# B&R Automation Studio project Parker_BMM_ST_V5_3147_V12 (part 32)

#### ClampR.ax
```
InitParameter (Version=5.06.1, NcSwId=ACP10)
  ACP10AXIS_typ:
    dig_in:
      level:
        reference = ncACTIV_HI
        pos_hw_end = ncACTIV_HI
        neg_hw_end = ncACTIV_HI
        trigger1 = ncACTIV_HI
        trigger2 = ncACTIV_HI + ncQUICKSTOP
    encoder_if:
      parameter:
        count_dir = ncSTANDARD
        scaling:
          load:
            units = 7087
            rev_motor = 5
    limit:
      parameter:
        v_pos = 70870.0  // Speed in positive direction    5600rpm 120000   4000rpm 85600
        v_neg = 70870.0
        a1_pos = 472400.0
        a2_pos = 472400.0
        a1_neg = 472400.0
        a2_neg = 472400.0
        t_jolt = 0.1
        t_in_pos = 0.0
        pos_sw_end = 8388607
        neg_sw_end = -8388608
        ds_warning = 354.0
        ds_stop = 708.0
        a_stop = 1.0E+30
        dv_stop = 0.0
        dv_stop_mode = ncOFF
    controller:
      mode = ncPOSITION
      position:
        kv = 66.0
        tn = 0.0
        t_predict = 0.0004
        t_total = 0.0004
        p_max = 1.0E+30
        i_max = 0.0
      speed:
        kv = 6.4
        tn = 0.1  // Integral action time 0.1
        t_filter = 0.0048  // Filter time constant 0.0048
        isq_filter1:
          type = ncOFF
          a0 = 0.0
          a1 = 0.0
          b0 = 0.0
          b1 = 0.0
          b2 = 0.0
          c0_par_id = 0
          c1_par_id = 0
        isq_filter2:
          type = ncOFF
          a0 = 0.0
          a1 = 0.0
          b0 = 0.0
          b1 = 0.0
          b2 = 0.0
          c0_par_id = 0
          c1_par_id = 0
        isq_filter3:
          type = ncOFF
          a0 = 0.0
          a1 = 0.0
          b0 = 0.0
          b1 = 0.0
          b2 = 0.0
          c0_par_id = 0
          c1_par_id = 0
      uf:
        type = ncLINEAR
        auto_config = ncMOTOR_PAR
        u0 = 0.0
        un = 0.0
        fn = 50.0
        k_f_slip = 0.0
      ff:
        mode = ncSTANDARD
        torque_load = 0.0
        torque_pos = 0.0
        torque_neg = 0.0
        kv_torque = 0.0
        inertia = 0.0
        t_filter_a = 0.0
      fb:
        mode = ncSTANDARD
        speed_mix_ratio = 0.0
        speed_kv = 2.0
      model:
        mass1:
          inertia = 0
          viscous_friction = 0
        mass2:
          inertia = 0
          viscous_friction = 0
          stiffness = 0
          damping = 0
    move:
      stop:
        parameter[0]:
          decel_ramp = ncA_LIMIT
          controller = ncON
        parameter[1]:
          decel_ramp = ncA_LIMIT
          controller = ncON
        parameter[2]:
          decel_ramp = ncA_LIMIT
          controller = ncON
        parameter[3]:
          decel_ramp = ncA_LIMIT
          controller = ncON
        quickstop:
          decel_ramp = ncA_LIMIT
          t_jolt = 0
        drive_error:
          decel_ramp = ncA_LIMIT
      homing:
        parameter:
          s = 0
          v_switch = 5000.0
          v_trigger = 500.0
          a = 50000.0
          mode = ncDIRECT
          edge_sw = ncPOSITIVE
          start_dir = ncPOSITIVE
          trigg_dir = ncPOSITIVE
          ref_pulse = ncOFF
          fix_dir = ncOFF
          tr_s_block = 0.0
          torque_lim = 0.0
          ds_block = 0.0
          ds_stop = 0.0
      basis:
        parameter:
          v_pos = 500.0
          v_neg = 500.0
          a1_pos = 5000.0
          a2_pos = 5000.0
          a1_neg = 5000.0
          a2_neg = 5000.0
    message:
      text:
        parameter:
          format = ncBREAK
          columns = 80
          data_modul = acp10etxen
```

### Data object Logical/Motion/init/ClampL (Ax)

#### ClampL.ax
```
InitParameter (Version=5.06.1, NcSwId=ACP10)
  ACP10AXIS_typ:
    dig_in:
      level:
        reference = ncACTIV_HI
        pos_hw_end = ncACTIV_HI
        neg_hw_end = ncACTIV_HI
        trigger1 = ncACTIV_HI
        trigger2 = ncACTIV_HI + ncQUICKSTOP
    encoder_if:
      parameter:
        count_dir = ncSTANDARD
        scaling:
          load:
            units = 1495
            rev_motor = 1
    limit:
      parameter:
        v_pos = 74750.0  // Speed in positive direction    5600rpm 120000   4000rpm 85600
        v_neg = 74750.0
        a1_pos = 747500.0
        a2_pos = 747500.0
        a1_neg = 747500.0
        a2_neg = 747500.0
        t_jolt = 0.1
        t_in_pos = 0.0
        pos_sw_end = 8388607
        neg_sw_end = -8388608
        ds_warning = 325.0
        ds_stop = 750.0
        a_stop = 1.0E+30
        dv_stop = 0.0
        dv_stop_mode = ncOFF
    controller:
      mode = ncPOSITION
      position:
        kv = 210.0
        tn = 0.0
        t_predict = 0.0004
        t_total = 0.0004
        p_max = 1.0E+30
        i_max = 0.0
      speed:
        kv = 15.0
        tn = 0.1  // Integral action time 0.1
        t_filter = 0.0048  // Filter time constant 0.0048
        isq_filter1:
          type = ncOFF
          a0 = 0.0
          a1 = 0.0
          b0 = 0.0
          b1 = 0.0
          b2 = 0.0
          c0_par_id = 0
          c1_par_id = 0
        isq_filter2:
          type = ncOFF
          a0 = 0.0
          a1 = 0.0
          b0 = 0.0
          b1 = 0.0
          b2 = 0.0
          c0_par_id = 0
          c1_par_id = 0
        isq_filter3:
          type = ncOFF
          a0 = 0.0
          a1 = 0.0
          b0 = 0.0
          b1 = 0.0
          b2 = 0.0
          c0_par_id = 0
          c1_par_id = 0
      uf:
        type = ncLINEAR
        auto_config = ncMOTOR_PAR
        u0 = 0.0
        un = 0.0
        fn = 50.0
        k_f_slip = 0.0
      ff:
        mode = ncSTANDARD
        torque_load = 0.0
        torque_pos = 0.0
        torque_neg = 0.0
        kv_torque = 0.0
        inertia = 0.0
        t_filter_a = 0.0
      fb:
        mode = ncSTANDARD
        speed_mix_ratio = 0.0
        speed_kv = 2.0
      model:
        mass1:
          inertia = 0
          viscous_friction = 0
        mass2:
          inertia = 0
          viscous_friction = 0
          stiffness = 0
          damping = 0
    move:
      stop:
        parameter[0]:
          decel_ramp = ncA_LIMIT
          controller = ncON
        parameter[1]:
          decel_ramp = ncA_LIMIT
          controller = ncON
        parameter[2]:
          decel_ramp = ncA_LIMIT
          controller = ncON
        parameter[3]:
          decel_ramp = ncA_LIMIT
          controller = ncON
        quickstop:
          decel_ramp = ncA_LIMIT
          t_jolt = 0
        drive_error:
          decel_ramp = ncA_LIMIT
      homing:
        parameter:
          s = 0
          v_switch = 5000.0
          v_trigger = 500.0
          a = 50000.0
          mode = ncDIRECT
          edge_sw = ncPOSITIVE
          start_dir = ncPOSITIVE
          trigg_dir = ncPOSITIVE
          ref_pulse = ncOFF
          fix_dir = ncOFF
          tr_s_block = 0.0
          torque_lim = 0.0
          ds_block = 0.0
          ds_stop = 0.0
      basis:
        parameter:
          v_pos = 500.0
          v_neg = 500.0
          a1_pos = 5000.0
          a2_pos = 5000.0
          a1_neg = 5000.0
          a2_neg = 5000.0
    message:
      text:
        parameter:
          format = ncBREAK
          columns = 80
          data_modul = acp10etxen
```

### Data object Logical/Motion/init/CarriageR (Ax)

#### CarriageR.ax
```
InitParameter (Version=5.06.1, NcSwId=ACP10)
  ACP10AXIS_typ:
    dig_in:
      level:
        reference = ncACTIV_HI
        pos_hw_end = ncACTIV_HI
        neg_hw_end = ncACTIV_HI
        trigger1 = ncACTIV_HI
        trigger2 = ncACTIV_HI + ncQUICKSTOP
    encoder_if:
      parameter:
        count_dir = ncSTANDARD
        scaling:
          load:
            units = 2571
            rev_motor = 2
    limit:
      parameter:
        v_pos = 96410.0
        v_neg = 96410.0
        a1_pos = 964100.0
        a2_pos = 964100.0
        a1_neg = 964100.0
        a2_neg = 964100.0
        t_jolt = 0.1
        t_in_pos = 0.0
        pos_sw_end = 8388607
        neg_sw_end = -8388608
        ds_warning = 320.0
        ds_stop = 640.0
        a_stop = 1.0E+30
        dv_stop = 0.0
        dv_stop_mode = ncOFF
    controller:
      mode = ncPOSITION
      position:
        kv = 190.0
        tn = 0.0
        t_predict = 0.0004
        t_total = 0.0004
        p_max = 1.0E+30
        i_max = 0.0
      speed:
        kv = 7.8
        tn = 0.0
        t_filter = 0.0
        isq_filter1:
          type = ncOFF
          a0 = 0.0
          a1 = 0.0
          b0 = 0.0
          b1 = 0.0
          b2 = 0.0
          c0_par_id = 0
          c1_par_id = 0
        isq_filter2:
          type = ncOFF
          a0 = 0.0
          a1 = 0.0
          b0 = 0.0
          b1 = 0.0
          b2 = 0.0
          c0_par_id = 0
          c1_par_id = 0
        isq_filter3:
          type = ncOFF
          a0 = 0.0
          a1 = 0.0
          b0 = 0.0
          b1 = 0.0
          b2 = 0.0
          c0_par_id = 0
          c1_par_id = 0
      uf:
        type = ncLINEAR
        auto_config = ncMOTOR_PAR
        u0 = 0.0
        un = 0.0
        fn = 50.0
        k_f_slip = 0.0
      ff:
        mode = ncSTANDARD
        torque_load = 0.0
        torque_pos = 0.0
        torque_neg = 0.0
        kv_torque = 0.0
        inertia = 0.0
        t_filter_a = 0.0
      fb:
        mode = ncSTANDARD
        speed_mix_ratio = 0.0
        speed_kv = 2.0
      model:
        mass1:
          inertia = 0
          viscous_friction = 0
        mass2:
          inertia = 0
          viscous_friction = 0
          stiffness = 0
          damping = 0
    move:
      stop:
        parameter[0]:
          decel_ramp = ncA_LIMIT
          controller = ncON
        parameter[1]:
          decel_ramp = ncA_LIMIT
          controller = ncON
        parameter[2]:
          decel_ramp = ncA_LIMIT
          controller = ncON
        parameter[3]:
          decel_ramp = ncA_LIMIT
          controller = ncON
        quickstop:
          decel_ramp = ncA_LIMIT
          t_jolt = 0
        drive_error:
          decel_ramp = ncA_LIMIT
      homing:
        parameter:
          s = 0
          v_switch = 5000.0
          v_trigger = 500.0
          a = 50000.0
          mode = ncDIRECT
          edge_sw = ncPOSITIVE
          start_dir = ncPOSITIVE
          trigg_dir = ncPOSITIVE
          ref_pulse = ncOFF
          fix_dir = ncOFF
          tr_s_block = 0.0
          torque_lim = 0.0
          ds_block = 0.0
          ds_stop = 0.0
      basis:
        parameter:
          v_pos = 5000.0
          v_neg = 5000.0
          a1_pos = 50000.0
          a2_pos = 50000.0
          a1_neg = 50000.0
          a2_neg = 50000.0
    message:
      text:
        parameter:
          format = ncBREAK
          columns = 80
          data_modul = acp10etxen
```

### Data object Logical/Motion/init/CarriageL (Ax)

#### CarriageL.ax
```
InitParameter (Version=5.06.1, NcSwId=ACP10)
  ACP10AXIS_typ:
    dig_in:
      level:
        reference = ncACTIV_HI
        pos_hw_end = ncACTIV_HI
        neg_hw_end = ncACTIV_HI
        trigger1 = ncACTIV_HI
        trigger2 = ncACTIV_HI + ncQUICKSTOP
    encoder_if:
      parameter:
        count_dir = ncSTANDARD
        scaling:
          load:
            units = 1433
            rev_motor = 1
    limit:
      parameter:
        v_pos = 107475.0
        v_neg = 107475.0
        a1_pos = 1074750.0
        a2_pos = 1074750.0
        a1_neg = 1074750.0
        a2_neg = 1074750.0
        t_jolt = 0.1
        t_in_pos = 0.0
        pos_sw_end = 8388607
        neg_sw_end = -8388608
        ds_warning = 716.0
        ds_stop = 360.0
        a_stop = 1.0E+30
        dv_stop = 0.0
        dv_stop_mode = ncOFF
    controller:
      mode = ncPOSITION
      position:
        kv = 50.0
        tn = 0.0
        t_predict = 0.0004
        t_total = 0.0004
        p_max = 1.0E+30
        i_max = 0.0
      speed:
        kv = 2.0
        tn = 0.0
        t_filter = 0.0
        isq_filter1:
          type = ncOFF
          a0 = 0.0
          a1 = 0.0
          b0 = 0.0
          b1 = 0.0
          b2 = 0.0
          c0_par_id = 0
          c1_par_id = 0
        isq_filter2:
          type = ncOFF
          a0 = 0.0
          a1 = 0.0
          b0 = 0.0
          b1 = 0.0
          b2 = 0.0
          c0_par_id = 0
          c1_par_id = 0
        isq_filter3:
          type = ncOFF
          a0 = 0.0
          a1 = 0.0
          b0 = 0.0
          b1 = 0.0
          b2 = 0.0
          c0_par_id = 0
          c1_par_id = 0
      uf:
        type = ncLINEAR
        auto_config = ncMOTOR_PAR
        u0 = 0.0
        un = 0.0
        fn = 50.0
        k_f_slip = 0.0
      ff:
        mode = ncSTANDARD
        torque_load = 0.0
        torque_pos = 0.0
        torque_neg = 0.0
        kv_torque = 0.0
        inertia = 0.0
        t_filter_a = 0.0
      fb:
        mode = ncSTANDARD
        speed_mix_ratio = 0.0
        speed_kv = 2.0
      model:
        mass1:
          inertia = 0
          viscous_friction = 0
        mass2:
          inertia = 0
          viscous_friction = 0
          stiffness = 0
          damping = 0
    move:
      stop:
        parameter[0]:
          decel_ramp = ncA_LIMIT
          controller = ncON
        parameter[1]:
          decel_ramp = ncA_LIMIT
          controller = ncON
        parameter[2]:
          decel_ramp = ncA_LIMIT
          controller = ncON
        parameter[3]:
          decel_ramp = ncA_LIMIT
          controller = ncON
        quickstop:
          decel_ramp = ncA_LIMIT
          t_jolt = 0
        drive_error:
          decel_ramp = ncA_LIMIT
      homing:
        parameter:
          s = 0
          v_switch = 5000.0
          v_trigger = 500.0
          a = 50000.0
          mode = ncDIRECT
          edge_sw = ncPOSITIVE
          start_dir = ncPOSITIVE
          trigg_dir = ncPOSITIVE
          ref_pulse = ncOFF
          fix_dir = ncOFF
          tr_s_block = 0.0
          torque_lim = 0.0
          ds_block = 0.0
          ds_stop = 0.0
      basis:
        parameter:
          v_pos = 1000.0
          v_neg = 1000.0
          a1_pos = 50000.0
          a2_pos = 50000.0
          a1_neg = 50000.0
          a2_neg = 50000.0
    message:
      text:
        parameter:
          format = ncBREAK
          columns = 80
          data_modul = acp10etxen
```

### Data object Logical/Motion/init/BlowPinR (Ax)

#### BlowPinR.ax
```
InitParameter (Version=5.06.1, NcSwId=ACP10)
  ACP10AXIS_typ:
    dig_in:
      level:
        reference = ncACTIV_HI
        pos_hw_end = ncACTIV_HI
        neg_hw_end = ncACTIV_HI
        trigger1 = ncACTIV_HI
        trigger2 = ncACTIV_HI + ncQUICKSTOP
    encoder_if:
      parameter:
        count_dir = ncSTANDARD
        scaling:
          load:
            units = 2000
            rev_motor = 1
    limit:
      parameter:
        v_pos = 65000.0
        v_neg = 65000.0
        a1_pos = 1500000.0
        a2_pos = 1500000.0
        a1_neg = 1500000.0
        a2_neg = 1500000.0
        t_jolt = 0.1
        t_in_pos = 0.0
        pos_sw_end = 8388607
        neg_sw_end = -8388608
        ds_warning = 500.0
        ds_stop = 1000.0
        a_stop = 1.0E+30
        dv_stop = 0.0
        dv_stop_mode = ncOFF
    controller:
      mode = ncPOSITION
      position:
        kv = 135.0
        tn = 0.0
        t_predict = 0.0004
        t_total = 0.0004
        p_max = 1.0E+30
        i_max = 0.0
      speed:
        kv = 1.0
        tn = 0.0
        t_filter = 0.0
        isq_filter1:
          type = ncOFF
          a0 = 0.0
          a1 = 0.0
          b0 = 0.0
          b1 = 0.0
          b2 = 0.0
          c0_par_id = 0
          c1_par_id = 0
        isq_filter2:
          type = ncOFF
          a0 = 0.0
          a1 = 0.0
          b0 = 0.0
          b1 = 0.0
          b2 = 0.0
          c0_par_id = 0
          c1_par_id = 0
        isq_filter3:
          type = ncOFF
          a0 = 0.0
          a1 = 0.0
          b0 = 0.0
          b1 = 0.0
          b2 = 0.0
          c0_par_id = 0
          c1_par_id = 0
      uf:
        type = ncLINEAR
        auto_config = ncMOTOR_PAR
        u0 = 0.0
        un = 0.0
        fn = 50.0
        k_f_slip = 0.0
      ff:
        mode = ncSTANDARD
        torque_load = 0.0
        torque_pos = 0.0
        torque_neg = 0.0
        kv_torque = 0.0
        inertia = 0.0
        t_filter_a = 0.0
      fb:
        mode = ncSTANDARD
        speed_mix_ratio = 0.0
        speed_kv = 0.0
      model:
        mass1:
          inertia = 0.0
          viscous_friction = 0.0
        mass2:
          inertia = 0.0
          viscous_friction = 0.0
          stiffness = 0.0
          damping = 0.0
    move:
      stop:
        parameter[0]:
          decel_ramp = ncA_LIMIT
          controller = ncON
        parameter[1]:
          decel_ramp = ncA_LIMIT
          controller = ncON
        parameter[2]:
          decel_ramp = ncA_LIMIT
          controller = ncON
        parameter[3]:
          decel_ramp = ncA_LIMIT
          controller = ncON
        quickstop:
          decel_ramp = ncA_LIMIT
          t_jolt = 0.0
        drive_error:
          decel_ramp = ncA_LIMIT
      homing:
        parameter:
          s = 0
          v_switch = 5000.0
          v_trigger = 500.0
          a = 50000.0
          mode = ncDIRECT
          edge_sw = ncPOSITIVE
          start_dir = ncPOSITIVE
          trigg_dir = ncPOSITIVE
          ref_pulse = ncOFF
          fix_dir = ncOFF
          tr_s_block = 0.0
          torque_lim = 0.0
          ds_block = 0.0
          ds_stop = 0.0
      basis:
        parameter:
          v_pos = 5000.0
          v_neg = 5000.0
          a1_pos = 50000.0
          a2_pos = 50000.0
          a1_neg = 50000.0
          a2_neg = 50000.0
    message:
      text:
        parameter:
          format = ncBREAK
          columns = 80
          data_modul = acp10etxen
```

### Data object Logical/Motion/init/BlowPinL (Ax)

#### BlowPinL.ax
```
InitParameter (Version=5.06.1, NcSwId=ACP10)
  ACP10AXIS_typ:
    dig_in:
      level:
        reference = ncACTIV_HI
        pos_hw_end = ncACTIV_HI
        neg_hw_end = ncACTIV_HI
        trigger1 = ncACTIV_HI
        trigger2 = ncACTIV_HI + ncQUICKSTOP
    encoder_if:
      parameter:
        count_dir = ncSTANDARD
        scaling:
          load:
            units = 2000
            rev_motor = 1
    limit:
      parameter:
        v_pos = 65000.0
        v_neg = 65000.0
        a1_pos = 1500000.0
        a2_pos = 1500000.0
        a1_neg = 1500000.0
        a2_neg = 1500000.0
        t_jolt = 0.1
        t_in_pos = 0.0
        pos_sw_end = 8388607
        neg_sw_end = -8388608
        ds_warning = 500.0
        ds_stop = 1000.0
        a_stop = 1.0E+30
        dv_stop = 0.0
        dv_stop_mode = ncOFF
    controller:
      mode = ncPOSITION
      position:
        kv = 170.0
        tn = 0.0
        t_predict = 0.0004
        t_total = 0.0004
        p_max = 1.0E+30
        i_max = 0.0
      speed:
        kv = 3.25
        tn = 0.0
        t_filter = 0.0
        isq_filter1:
          type = ncOFF
          a0 = 0.0
          a1 = 0.0
          b0 = 0.0
          b1 = 0.0
          b2 = 0.0
          c0_par_id = 0
          c1_par_id = 0
        isq_filter2:
          type = ncOFF
          a0 = 0.0
          a1 = 0.0
          b0 = 0.0
          b1 = 0.0
          b2 = 0.0
          c0_par_id = 0
          c1_par_id = 0
        isq_filter3:
          type = ncOFF
          a0 = 0.0
          a1 = 0.0
          b0 = 0.0
          b1 = 0.0
          b2 = 0.0
          c0_par_id = 0
          c1_par_id = 0
      uf:
        type = ncLINEAR
        auto_config = ncMOTOR_PAR
        u0 = 0.0
        un = 0.0
        fn = 50.0
        k_f_slip = 0.0
      ff:
        mode = ncSTANDARD
        torque_load = 0.0
        torque_pos = 0.0
        torque_neg = 0.0
        kv_torque = 0.0
        inertia = 0.0
        t_filter_a = 0.0
      fb:
        mode = ncSTANDARD
        speed_mix_ratio = 0.0
        speed_kv = 2.0
      model:
        mass1:
          inertia = 0
          viscous_friction = 0
        mass2:
          inertia = 0
          viscous_friction = 0
          stiffness = 0
          damping = 0
    move:
      stop:
        parameter[0]:
          decel_ramp = ncA_LIMIT
          controller = ncON
        parameter[1]:
          decel_ramp = ncA_LIMIT
          controller = ncON
        parameter[2]:
          decel_ramp = ncA_LIMIT
          controller = ncON
        parameter[3]:
          decel_ramp = ncA_LIMIT
          controller = ncON
        quickstop:
          decel_ramp = ncA_LIMIT
          t_jolt = 0
        drive_error:
          decel_ramp = ncA_LIMIT
      homing:
        parameter:
          s = 0
          v_switch = 5000.0
          v_trigger = 500.0
          a = 50000.0
          mode = ncDIRECT
          edge_sw = ncPOSITIVE
          start_dir = ncPOSITIVE
          trigg_dir = ncPOSITIVE
          ref_pulse = ncOFF
          fix_dir = ncOFF
          tr_s_block = 0.0
          torque_lim = 0.0
          ds_block = 0.0
          ds_stop = 0.0
      basis:
        parameter:
          v_pos = 500.0
          v_neg = 500.0
          a1_pos = 50000.0
          a2_pos = 50000.0
          a1_neg = 50000.0
          a2_neg = 50000.0
    message:
      text:
        parameter:
          format = ncBREAK
          columns = 80
          data_modul = acp10etxen
```

### Data object Logical/Motion/init/BlowPin2R (Ax)

#### BlowPinR.ax
```
InitParameter (Version=5.06.1, NcSwId=ACP10)
  ACP10AXIS_typ:
    dig_in:
      level:
        reference = ncACTIV_HI
        pos_hw_end = ncACTIV_HI
        neg_hw_end = ncACTIV_HI
        trigger1 = ncACTIV_HI
        trigger2 = ncACTIV_HI + ncQUICKSTOP
    encoder_if:
      parameter:
        count_dir = ncSTANDARD
        scaling:
          load:
            units = 2000
            rev_motor = 1
    limit:
      parameter:
        v_pos = 65000.0
        v_neg = 65000.0
        a1_pos = 1500000.0
        a2_pos = 1500000.0
        a1_neg = 1500000.0
        a2_neg = 1500000.0
        t_jolt = 0.1
        t_in_pos = 0.0
        pos_sw_end = 8388607
        neg_sw_end = -8388608
        ds_warning = 500.0
        ds_stop = 1000.0
        a_stop = 1.0E+30
        dv_stop = 0.0
        dv_stop_mode = ncOFF
    controller:
      mode = ncPOSITION
      position:
        kv = 213.0
        tn = 0.0
        t_predict = 0.0004
        t_total = 0.0004
        p_max = 1.0E+30
        i_max = 0.0
      speed:
        kv = 2.7
        tn = 0.0
        t_filter = 0.0
        isq_filter1:
          type = ncOFF
          a0 = 0.0
          a1 = 0.0
          b0 = 0.0
          b1 = 0.0
          b2 = 0.0
          c0_par_id = 0
          c1_par_id = 0
        isq_filter2:
          type = ncOFF
          a0 = 0.0
          a1 = 0.0
          b0 = 0.0
          b1 = 0.0
          b2 = 0.0
          c0_par_id = 0
          c1_par_id = 0
        isq_filter3:
          type = ncOFF
          a0 = 0.0
          a1 = 0.0
          b0 = 0.0
          b1 = 0.0
          b2 = 0.0
          c0_par_id = 0
          c1_par_id = 0
      uf:
        type = ncLINEAR
        auto_config = ncMOTOR_PAR
        u0 = 0.0
        un = 0.0
        fn = 50.0
        k_f_slip = 0.0
      ff:
        mode = ncSTANDARD
        torque_load = 0.0
        torque_pos = 0.0
        torque_neg = 0.0
        kv_torque = 0.0
        inertia = 0.0
        t_filter_a = 0.0
      fb:
        mode = ncSTANDARD
        speed_mix_ratio = 0.0
        speed_kv = 0.0
      model:
        mass1:
          inertia = 0.0
          viscous_friction = 0.0
        mass2:
          inertia = 0.0
          viscous_friction = 0.0
          stiffness = 0.0
          damping = 0.0
    move:
      stop:
        parameter[0]:
          decel_ramp = ncA_LIMIT
          controller = ncON
        parameter[1]:
          decel_ramp = ncA_LIMIT
          controller = ncON
        parameter[2]:
          decel_ramp = ncA_LIMIT
          controller = ncON
        parameter[3]:
          decel_ramp = ncA_LIMIT
          controller = ncON
        quickstop:
          decel_ramp = ncA_LIMIT
          t_jolt = 0.0
        drive_error:
          decel_ramp = ncA_LIMIT
      homing:
        parameter:
          s = 0
          v_switch = 5000.0
          v_trigger = 500.0
          a = 50000.0
          mode = ncDIRECT
          edge_sw = ncPOSITIVE
          start_dir = ncPOSITIVE
          trigg_dir = ncPOSITIVE
          ref_pulse = ncOFF
          fix_dir = ncOFF
          tr_s_block = 0.0
          torque_lim = 0.0
          ds_block = 0.0
          ds_stop = 0.0
      basis:
        parameter:
          v_pos = 1000.0
          v_neg = 1000.0
          a1_pos = 1000.0
          a2_pos = 1000.0
          a1_neg = 1000.0
          a2_neg = 1000.0
    message:
      text:
        parameter:
          format = ncBREAK
          columns = 80
          data_modul = acp10etxen
```

- Data object Logical/Motion/init/BlowPin2L (Ax) (no source held here)

### Data object Logical/Motion/init/Power (Ax)

#### Power.ax
```
InitParameter (Version=2.48.1, NcSwId=Acp10)
  ACP10AXIS_typ:
    dig_in:
      level:
        reference = ncACTIV_HI
        pos_hw_end = ncACTIV_HI
        neg_hw_end = ncACTIV_HI
        trigger1 = ncACTIV_HI
        trigger2 = ncACTIV_HI + ncQUICKSTOP
    encoder_if:
      parameter:
        count_dir = ncSTANDARD
        scaling:
          load:
            units = 1000
            rev_motor = 1
    limit:
      parameter:
        v_pos = 10000
        v_neg = 10000
        a1_pos = 50000
        a2_pos = 50000
        a1_neg = 50000
        a2_neg = 50000
        t_jolt = 0
        t_in_pos = 0
        pos_sw_end = 2000000000
        neg_sw_end = -2000000000
        ds_warning = 500
        ds_stop = 1000
        a_stop = 1.0e30
        dv_stop = 0
        dv_stop_mode = ncOFF
    controller:
      mode = ncPOSITION
      position:
        kv = 50
        tn = 0
        t_predict = 0.0004
        t_total = 0.0004
        p_max = 1.0e30
        i_max = 0
      speed:
        kv = 2.0
        tn = 0
        t_filter = 0.0
        isq_filter1:
          type = ncOFF
          a0 = 0.0
          a1 = 0.0
          b0 = 0.0
          b1 = 0.0
          b2 = 0.0
          c0_par_id = 0
          c1_par_id = 0
        isq_filter2:
          type = ncOFF
          a0 = 0.0
          a1 = 0.0
          b0 = 0.0
          b1 = 0.0
          b2 = 0.0
          c0_par_id = 0
          c1_par_id = 0
        isq_filter3:
          type = ncOFF
          a0 = 0.0
          a1 = 0.0
          b0 = 0.0
          b1 = 0.0
          b2 = 0.0
          c0_par_id = 0
          c1_par_id = 0
      uf:
        type = ncLINEAR
        auto_config = ncMOTOR_PAR
        u0 = 0
        un = 0
        fn = 50.0
        k_f_slip = 0
      ff:
        torque_load = 0.0
        torque_pos = 0.0
        torque_neg = 0.0
        kv_torque = 0.0
        inertia = 0.0
        t_filter_a = 0.0
    move:
      stop:
        parameter[0]:
          decel_ramp = ncA_LIMIT
          controller = ncON
        parameter[1]:
          decel_ramp = ncA_LIMIT
          controller = ncON
        parameter[2]:
          decel_ramp = ncA_LIMIT
          controller = ncON
        parameter[3]:
          decel_ramp = ncA_LIMIT
          controller = ncON
        quickstop:
          decel_ramp = ncA_LIMIT
        drive_error:
          decel_ramp = ncA_LIMIT
      homing:
        parameter:
          s = 0
          v_switch = 5000
          v_trigger = 500
          a = 50000
          mode = ncDIRECT
          edge_sw = ncPOSITIVE
          start_dir = ncPOSITIVE
          trigg_dir = ncPOSITIVE
          ref_pulse = ncOFF
          fix_dir = ncOFF
          tr_s_block = 0
          torque_lim = 0
          ds_block = 0
          ds_stop = 0
      basis:
        parameter:
          v_pos = 5000
          v_neg = 5000
          a1_pos = 50000
          a2_pos = 50000
          a1_neg = 50000
          a2_neg = 50000
    message:
      text:
        parameter:
          format = ncBREAK
          columns = 80
          data_modul = acp10etxen
```

### Data object Logical/Motion/init/ExtrLift (Ax)

#### ExtrLift.ax
```
InitParameter (Version=5.06.1, NcSwId=ACP10)
  ACP10AXIS_typ:
    dig_in:
      level:
        reference = ncACTIV_HI
        pos_hw_end = ncACTIV_HI
        neg_hw_end = ncACTIV_HI
        trigger1 = ncACTIV_HI
        trigger2 = ncACTIV_HI + ncQUICKSTOP
    encoder_if:
      parameter:
        count_dir = ncSTANDARD
        scaling:
          load:
            units = 5733  // Units at the load  16992
            rev_motor = 5  // Motor revolutions 10
    limit:
      parameter:
        v_pos = 10000.0  // Speed in positive direction 3000rpm =933333  6000rpm = 1866666  7200rpm= 2240000  
        v_neg = 5000.0
        a1_pos = 20000.0
        a2_pos = 20000.0
        a1_neg = 20000.0
        a2_neg = 20000.0
        t_jolt = 0.1
        t_in_pos = 0
        pos_sw_end = 2000000000
        neg_sw_end = -2000000000
        ds_warning = 286.0
        ds_stop = 573.0
        a_stop = 1.0e30
        dv_stop = 0
        dv_stop_mode = ncOFF
    controller:
      mode = ncPOSITION
      position:
        kv = 250.0
        tn = 0
        t_predict = 0.0004
        t_total = 0.0004
        p_max = 1.0E+30
        i_max = 0
      speed:
        kv = 4.0
        tn = 0.1
        t_filter = 0.0
        isq_filter1:
          type = ncOFF
          a0 = 0.0
          a1 = 0.0
          b0 = 0.0
          b1 = 0.0
          b2 = 0.0
          c0_par_id = 0
          c1_par_id = 0
        isq_filter2:
          type = ncOFF
          a0 = 0.0
          a1 = 0.0
          b0 = 0.0
          b1 = 0.0
          b2 = 0.0
          c0_par_id = 0
          c1_par_id = 0
        isq_filter3:
          type = ncOFF
          a0 = 0.0
          a1 = 0.0
          b0 = 0.0
          b1 = 0.0
          b2 = 0.0
          c0_par_id = 0
          c1_par_id = 0
      uf:
        type = ncLINEAR
        auto_config = ncMOTOR_PAR
        u0 = 0
        un = 0
        fn = 50.0
        k_f_slip = 0
      ff:
        mode = ncSTANDARD
        torque_load = 0.0
        torque_pos = 0.0
        torque_neg = 0.0
        kv_torque = 0.0
        inertia = 0.0
        t_filter_a = 0.0
      fb:
        mode = ncSTANDARD
        speed_mix_ratio = 0.0
        speed_kv = 2.0
      model:
        mass1:
          inertia = 0
          viscous_friction = 0
        mass2:
          inertia = 0
          viscous_friction = 0
          stiffness = 0
          damping = 0
    move:
      stop:
        parameter[0]:
          decel_ramp = ncA_LIMIT
          controller = ncON
        parameter[1]:
          decel_ramp = ncA_LIMIT
          controller = ncON
        parameter[2]:
          decel_ramp = ncA_LIMIT
          controller = ncON
        parameter[3]:
          decel_ramp = ncA_LIMIT
          controller = ncON
        quickstop:
          decel_ramp = ncA_LIMIT
          t_jolt = 0
        drive_error:
          decel_ramp = ncA_LIMIT
      homing:
        parameter:
          s = 0
          v_switch = 5000.0
          v_trigger = 500.0
          a = 50000.0
          mode = ncDIRECT
          edge_sw = ncPOSITIVE
          start_dir = ncPOSITIVE
          trigg_dir = ncPOSITIVE
          ref_pulse = ncOFF
          fix_dir = ncOFF
          tr_s_block = 0
          torque_lim = 0
          ds_block = 0
          ds_stop = 0
      basis:
        parameter:
          v_pos = 5000
          v_neg = 5000
          a1_pos = 50000
          a2_pos = 50000
          a1_neg = 50000
          a2_neg = 50000
    message:
      text:
        parameter:
          format = ncBREAK
          columns = 80
          data_modul = acp10etxen
```

### Data object Logical/Motion/init/ThickInit (Ax)

#### ThickInit.ax
```
InitParameter (Version=5.06.1, NcSwId=ACP10)
  ACP10AXIS_typ:
    dig_in:
      level:
        reference = ncACTIV_HI
        pos_hw_end = ncACTIV_HI
        neg_hw_end = ncACTIV_HI
        trigger1 = ncACTIV_HI
        trigger2 = ncACTIV_HI + ncQUICKSTOP
    encoder_if:
      parameter:
        count_dir = ncINVERSE
        scaling:
          load:
            units = 500
            rev_motor = 1
    limit:
      parameter:
        v_pos = 25000.0  // Speed in positive direction 
        v_neg = 25000.0
        a1_pos = 125000.0  // Acceleration in positive direction 
        a2_pos = 125000.0
        a1_neg = 125000.0
        a2_neg = 125000.0
        t_jolt = 0.1
        t_in_pos = 0.0
        pos_sw_end = 8388607
        neg_sw_end = -8388608
        ds_warning = 125.0
        ds_stop = 250.0
        a_stop = 1.0E+30
        dv_stop = 0.0
        dv_stop_mode = ncOFF
    controller:
      mode = ncPOSITION
      position:
        kv = 330.0
        tn = 0.0
        t_predict = 0.0004
        t_total = 0.0004
        p_max = 1.0E+30
        i_max = 0.0
      speed:
        kv = 11.4
        tn = 0.0
        t_filter = 0.0
        isq_filter1:
          type = ncOFF
          a0 = 0.0
          a1 = 0.0
          b0 = 0.0
          b1 = 0.0
          b2 = 0.0
          c0_par_id = 0
          c1_par_id = 0
        isq_filter2:
          type = ncOFF
          a0 = 0.0
          a1 = 0.0
          b0 = 0.0
          b1 = 0.0
          b2 = 0.0
          c0_par_id = 0
          c1_par_id = 0
        isq_filter3:
          type = ncOFF
          a0 = 0.0
          a1 = 0.0
          b0 = 0.0
          b1 = 0.0
          b2 = 0.0
          c0_par_id = 0
          c1_par_id = 0
      uf:
        type = ncLINEAR
        auto_config = ncMOTOR_PAR
        u0 = 0.0
        un = 0.0
        fn = 50.0
        k_f_slip = 0.0
      ff:
        mode = ncSTANDARD
        torque_load = 0.0
        torque_pos = 0.0
        torque_neg = 0.0
        kv_torque = 0.0
        inertia = 0.0
        t_filter_a = 0.0
      fb:
        mode = ncSTANDARD
        speed_mix_ratio = 0.0
        speed_kv = 2.0
      model:
        mass1:
          inertia = 0
          viscous_friction = 0
        mass2:
          inertia = 0
          viscous_friction = 0
          stiffness = 0
          damping = 0
    move:
      stop:
        parameter[0]:
          decel_ramp = ncA_LIMIT
          controller = ncON
        parameter[1]:
          decel_ramp = ncA_LIMIT
          controller = ncON
        parameter[2]:
          decel_ramp = ncA_LIMIT
          controller = ncON
        parameter[3]:
          decel_ramp = ncA_LIMIT
          controller = ncON
        quickstop:
          decel_ramp = ncA_LIMIT
          t_jolt = 0
        drive_error:
          decel_ramp = ncA_LIMIT
      homing:
        parameter:
          s = 0
          v_switch = 5000.0
          v_trigger = 500.0
          a = 50000.0
          mode = ncDIRECT
          edge_sw = ncPOSITIVE
          start_dir = ncPOSITIVE
          trigg_dir = ncPOSITIVE
          ref_pulse = ncOFF
          fix_dir = ncOFF
          tr_s_block = 0.0
          torque_lim = 0.0
          ds_block = 0.0
          ds_stop = 0.0
      basis:
        parameter:
          v_pos = 2000.0
          v_neg = 2000.0
          a1_pos = 40000.0
          a2_pos = 40000.0
          a1_neg = 40000.0
          a2_neg = 40000.0
    message:
      text:
        parameter:
          format = ncBREAK
          columns = 80
          data_modul = acp10etxen
```

### Data object Logical/Motion/para/Tansfer (Apt)

#### Transfer.apt
```
AcoposParameterTable:
  Root Parameters:
    Configure Parameter:
      128 = 1 (Name=SGEN_SW_END_IGNORE)  // Limit values: Ignore SW end positions
      300 = 300 (Name=UDC_DETECTION, Unit=V, Disabled=FALSE)  // CTRL DC bus: Voltage detection: Lower limit
      80 = 1 (Name=PHASE_MON_IGNORE, Disabled=TRUE)  // Power mains: Ignore phase failure
    VAR_XX_X+0:
      777 = VAR_I4_0+0 (Name=FUNCTION_BLOCK_CREATE)  // VAR_XX_X+0
      VAR_R4_X_0:
        4128 = 0.0 (Name=VAR_R4_0+0)
        4136 = 0.0 (Name=VAR_R4_1+0)
        4144 = 0.142 (Name=VAR_R4_2+0)  // temp junction Kp
        4152 = 0.142 (Name=VAR_R4_3+0)  // temp motor Kp
      VAR_I4_X_0 (Disabled=FALSE)
        4160 = 0.0 (Name=VAR_I2_0+0, Disabled=FALSE)  // FB0 FB VAR: Variable0 I2
        4168 = 0.0 (Name=VAR_I2_1+0, Disabled=FALSE)  // FB0 FB VAR: Variable1 I2
        4176 = 0.0 (Name=VAR_I2_2+0, Disabled=FALSE)  // FB0 FB VAR: Variable2 I2
        4184 = 0.0 (Name=VAR_I2_3+0, Disabled=FALSE)  // FB0 FB VAR: Variable3 I2
    Torque Limitation (Disabled=FALSE)
      Function Create (Disabled=FALSE)
        777 = ARITH_MODE+0 (Name=FUNCTION_BLOCK_CREATE, Disabled=FALSE)  // ARITH_0
        777 = ARITH_MODE+1 (Name=FUNCTION_BLOCK_CREATE, Disabled=FALSE)  // ARITH_1
        777 = ARITH_MODE+2 (Name=FUNCTION_BLOCK_CREATE, Disabled=FALSE)  // ARITH_2
        777 = ARITH_MODE+3 (Name=FUNCTION_BLOCK_CREATE, Disabled=FALSE)  // ARITH_3
        777 = ARITH_MODE+4 (Name=FUNCTION_BLOCK_CREATE, Disabled=FALSE)  // ARITH_4
        777 = ARITH_MODE+5 (Name=FUNCTION_BLOCK_CREATE, Disabled=FALSE)  // ARITH_5
        777 = MINMAX_MODE+0 (Name=FUNCTION_BLOCK_CREATE, Disabled=FALSE)  // MINMAX_0
        777 = MINMAX_MODE+1 (Name=FUNCTION_BLOCK_CREATE, Disabled=FALSE)  // MINMAX_1
        777 = EVWR_MODE+2 (Name=FUNCTION_BLOCK_CREATE, Disabled=FALSE)  // EVWR_2
        777 = EVWR_MODE+3 (Name=FUNCTION_BLOCK_CREATE, Disabled=FALSE)  // EVWR_3
        777 = EVWR_MODE+4 (Name=FUNCTION_BLOCK_CREATE, Disabled=FALSE)  // EVWR_4
        777 = EVWR_MODE+5 (Name=FUNCTION_BLOCK_CREATE, Disabled=FALSE)  // EVWR_5
      ARITH + 0 (Disabled=FALSE)
        3592 = TEMP_JUNCTION_LIM (Name=ARITH_IN1_PARID+0, Disabled=FALSE)  // TEMP_JUNCTION_LIM -- 842
        3600 = TEMP_JUNCTION (Name=ARITH_IN2_PARID+0, Disabled=FALSE)  // TEMP_JUNCTION -- 382
        3632 = 0 (Name=ARITH_K1+0, Disabled=FALSE)  // FB0 FB ARITH: Multiplication factor1
        3640 = 0 (Name=ARITH_K2+0, Disabled=FALSE)  // FB0 FB ARITH: Multiplication factor2
        3584 = 2 (Name=ARITH_MODE+0, Disabled=FALSE)  // y= x1 - x2
      ARITH + 1 (Disabled=FALSE)
        3593 = ARITH_VALUE_R4+0 (Name=ARITH_IN1_PARID+1, Disabled=FALSE)  // 3624
        3601 = VAR_R4_2+0 (Name=ARITH_IN2_PARID+1, Disabled=FALSE)  // 4144
        3633 = 0 (Name=ARITH_K1+1, Disabled=FALSE)  // FB1 FB ARITH: Multiplication factor1
        3641 = 0 (Name=ARITH_K2+1, Disabled=FALSE)  // FB1 FB ARITH: Multiplication factor2
        3585 = 3 (Name=ARITH_MODE+1, Disabled=FALSE)  // y = x1 * x2
      ARITH + 2 (Disabled=FALSE)
        3594 = MOTOR_TORQ_RATED (Name=ARITH_IN1_PARID+2, Disabled=FALSE)  // MOTOR_TORQ_RATED -- 53
        3602 = ARITH_VALUE_R4+1 (Name=ARITH_IN2_PARID+2, Disabled=FALSE)  // 3625
        3634 = 0 (Name=ARITH_K1+2, Disabled=FALSE)  // FB2 FB ARITH: Multiplication factor1
        3642 = 0 (Name=ARITH_K2+2, Disabled=FALSE)  // FB2 FB ARITH: Multiplication factor2
        3586 = 1 (Name=ARITH_MODE+2, Disabled=FALSE)  // y = x1 + x2
      ARITH + 3 (Disabled=FALSE)
        3595 = MOTOR_WIND_TEMP_MAX (Name=ARITH_IN1_PARID+3, Disabled=FALSE)  // 74 - MOTOR_WIND_TEMP_MAX
        3603 = TEMP_MOTOR (Name=ARITH_IN2_PARID+3, Disabled=FALSE)  // 381 - TEMP_MOTOR
        3635 = 0 (Name=ARITH_K1+3, Disabled=FALSE)  // FB3 FB ARITH: Multiplication factor1
        3643 = 0 (Name=ARITH_K2+3, Disabled=FALSE)  // FB3 FB ARITH: Multiplication factor2
        3587 = 2 (Name=ARITH_MODE+3, Disabled=FALSE)  // y = x1 - x2
      ARITH + 4 (Disabled=FALSE)
        3596 = ARITH_VALUE_R4+3 (Name=ARITH_IN1_PARID+4, Disabled=FALSE)  // 3627
        3604 = VAR_R4_3+0 (Name=ARITH_IN2_PARID+4, Disabled=FALSE)  // 4152
        3636 = 0 (Name=ARITH_K1+4, Disabled=FALSE)  // FB4 FB ARITH: Multiplication factor1
        3644 = 0 (Name=ARITH_K2+4, Disabled=FALSE)  // FB4 FB ARITH: Multiplication factor2
        3588 = 3 (Name=ARITH_MODE+4, Disabled=FALSE)  // y = x1 * x2
      ARITH + 5 (Disabled=FALSE)
        3597 = MOTOR_TORQ_RATED (Name=ARITH_IN1_PARID+5, Disabled=FALSE)  // MOTOR_TORQ_RATED -- 53
        3605 = ARITH_VALUE_R4+4 (Name=ARITH_IN2_PARID+5, Disabled=FALSE)  // 3628
        3637 = 0 (Name=ARITH_K1+5, Disabled=FALSE)  // FB5 FB ARITH: Multiplication factor1
        3645 = 0 (Name=ARITH_K2+5, Disabled=FALSE)  // FB5 FB ARITH: Multiplication factor2
        3589 = 1 (Name=ARITH_MODE+5, Disabled=FALSE)  // y = x1 + x2
      MINMAX + 0 (Disabled=FALSE)
        12312 = MOTOR_TORQ_MAX (Name=MINMAX_IN1_PARID+0, Disabled=FALSE)  // MOTOR_TORQ_MAX -- 54
        12320 = ARITH_VALUE_R4+2 (Name=MINMAX_IN2_PARID+0, Disabled=FALSE)  // 3626
        12328 = ARITH_VALUE_R4+5 (Name=MINMAX_IN3_PARID+0, Disabled=FALSE)  // 3629
        12288 = 1 (Name=MINMAX_MODE+0, Disabled=FALSE)  // MIN(MOTOR_TORQ_MAX,ARITH_VALUE_R4+1)
      MINMAX + 1 (Disabled=FALSE)
        12313 = VAR_R4_0+0 (Name=MINMAX_IN1_PARID+1, Disabled=FALSE)  // zero
        12321 = MINMAX_VALUE_R4+0 (Name=MINMAX_IN2_PARID+1, Disabled=FALSE)  // FB1 FB MINMAX: Parameter ID of input2
        12289 = 2 (Name=MINMAX_MODE+1, Disabled=FALSE)  // MAX(VAR_R4_0+0,MINMAX_VALUE_R4+0)
      EVWR + 2 (Disabled=FALSE)
        4610 = CONST_I4_ONE (Name=EVWR_EVENT_PARID+2, Disabled=FALSE)  // FB2 FB EVWR: Parameter ID of event input
        4618 = MINMAX_VALUE_R4+1 (Name=EVWR_IN_PARID+2, Disabled=FALSE)  // FB2 FB EVWR: Parameter ID of input
        4626 = 1 (Name=EVWR_EVENT_LEVEL+2, Disabled=FALSE)  // FB2 FB EVWR: Event level
        4634 = LIM_T2_POS (Name=EVWR_WR_PARID+2, Disabled=FALSE)  // 348
        4642 = 2 (Name=EVWR_MODE+2, Disabled=FALSE)  // mode - cyclic write
      EVWR + 3 (Disabled=FALSE)
        4611 = CONST_I4_ONE (Name=EVWR_EVENT_PARID+3, Disabled=FALSE)  // FB3 FB EVWR: Parameter ID of event input
        4619 = MINMAX_VALUE_R4+1 (Name=EVWR_IN_PARID+3, Disabled=FALSE)  // FB3 FB EVWR: Parameter ID of input
        4627 = 1 (Name=EVWR_EVENT_LEVEL+3, Disabled=FALSE)  // FB3 FB EVWR: Event level
        4635 = LIM_T2_NEG (Name=EVWR_WR_PARID+3, Disabled=FALSE)  // 349
        4643 = 2 (Name=EVWR_MODE+3, Disabled=FALSE)  // mode - cyclic write
      EVWR + 4 (Disabled=FALSE)
        4612 = CONST_I4_ONE (Name=EVWR_EVENT_PARID+4, Disabled=FALSE)  // FB4 FB EVWR: Parameter ID of event input
        4620 = MINMAX_VALUE_R4+1 (Name=EVWR_IN_PARID+4, Disabled=FALSE)  // FB4 FB EVWR: Parameter ID of input
        4628 = 1 (Name=EVWR_EVENT_LEVEL+4, Disabled=FALSE)  // FB4 FB EVWR: Event level
        4636 = LIM_T1_POS (Name=EVWR_WR_PARID+4, Disabled=FALSE)  // 248
        4644 = 2 (Name=EVWR_MODE+4, Disabled=FALSE)  // mode - cyclic write
      EVWR + 5 (Disabled=FALSE)
        4613 = CONST_I4_ONE (Name=EVWR_EVENT_PARID+5, Disabled=FALSE)  // FB5 FB EVWR: Parameter ID of event input
        4621 = MINMAX_VALUE_R4+1 (Name=EVWR_IN_PARID+5, Disabled=FALSE)  // FB5 FB EVWR: Parameter ID of input
        4629 = 1 (Name=EVWR_EVENT_LEVEL+5, Disabled=FALSE)  // FB5 FB EVWR: Event level
        4637 = LIM_T1_NEG (Name=EVWR_WR_PARID+5, Disabled=FALSE)  // 249
        4645 = 2 (Name=EVWR_MODE+5, Disabled=FALSE)  // mode - cyclic write
    HardWare Limit  For ACOPOS Multi:
      945 = VAR_I2_0+0 (Name=POS_LIMIT_SWITCH_PARID)  // Digital inputs: Parameter ID for positive end switch
      946 = VAR_I2_1+0 (Name=NEG_LIMIT_SWITCH_PARID)  // Digital inputs: Parameter ID for negative end switch
```

### Data object Logical/Motion/para/UpDn (Apt)

#### UpDn.apt
```
AcoposParameterTable:
  Root Parameters:
    Configure Parameter:
      128 = 1 (Name=SGEN_SW_END_IGNORE)  // Limit values: Ignore SW end positions
      80 = 1 (Name=PHASE_MON_IGNORE, Disabled=FALSE)  // Power mains: Ignore phase failure
    VAR_XX_X+0:
      777 = VAR_I4_0+0 (Name=FUNCTION_BLOCK_CREATE)  // VAR_XX_X+0
      VAR_R4_X_0:
        4128 = 0.0 (Name=VAR_R4_0+0)
        4136 = 0.0 (Name=VAR_R4_1+0)
        4144 = 0.3 (Name=VAR_R4_2+0)  // temp junction Kp
        4152 = 0.3 (Name=VAR_R4_3+0)  // temp motor Kp
    Torque Limitation (Disabled=FALSE)
      Function Create (Disabled=FALSE)
        777 = ARITH_MODE+0 (Name=FUNCTION_BLOCK_CREATE, Disabled=FALSE)  // ARITH_0
        777 = ARITH_MODE+1 (Name=FUNCTION_BLOCK_CREATE, Disabled=FALSE)  // ARITH_1
        777 = ARITH_MODE+2 (Name=FUNCTION_BLOCK_CREATE, Disabled=FALSE)  // ARITH_2
        777 = ARITH_MODE+3 (Name=FUNCTION_BLOCK_CREATE, Disabled=FALSE)  // ARITH_3
        777 = ARITH_MODE+4 (Name=FUNCTION_BLOCK_CREATE, Disabled=FALSE)  // ARITH_4
        777 = ARITH_MODE+5 (Name=FUNCTION_BLOCK_CREATE, Disabled=FALSE)  // ARITH_5
        777 = MINMAX_MODE+0 (Name=FUNCTION_BLOCK_CREATE, Disabled=FALSE)  // MINMAX_0
        777 = MINMAX_MODE+1 (Name=FUNCTION_BLOCK_CREATE, Disabled=FALSE)  // MINMAX_1
        777 = EVWR_MODE+2 (Name=FUNCTION_BLOCK_CREATE, Disabled=FALSE)  // EVWR_2
        777 = EVWR_MODE+3 (Name=FUNCTION_BLOCK_CREATE, Disabled=FALSE)  // EVWR_3
        777 = EVWR_MODE+4 (Name=FUNCTION_BLOCK_CREATE, Disabled=FALSE)  // EVWR_4
        777 = EVWR_MODE+5 (Name=FUNCTION_BLOCK_CREATE, Disabled=FALSE)  // EVWR_5
      ARITH + 0 (Disabled=FALSE)
        3592 = TEMP_JUNCTION_LIM (Name=ARITH_IN1_PARID+0, Disabled=FALSE)  // TEMP_JUNCTION_LIM -- 842
        3600 = TEMP_JUNCTION (Name=ARITH_IN2_PARID+0, Disabled=FALSE)  // TEMP_JUNCTION -- 382
        3632 = 0 (Name=ARITH_K1+0, Disabled=FALSE)  // FB0 FB ARITH: Multiplication factor1
        3640 = 0 (Name=ARITH_K2+0, Disabled=FALSE)  // FB0 FB ARITH: Multiplication factor2
        3584 = 2 (Name=ARITH_MODE+0, Disabled=FALSE)  // y= x1 - x2
      ARITH + 1 (Disabled=FALSE)
        3593 = ARITH_VALUE_R4+0 (Name=ARITH_IN1_PARID+1, Disabled=FALSE)  // 3624
        3601 = VAR_R4_2+0 (Name=ARITH_IN2_PARID+1, Disabled=FALSE)  // 4144
        3633 = 0 (Name=ARITH_K1+1, Disabled=FALSE)  // FB1 FB ARITH: Multiplication factor1
        3641 = 0 (Name=ARITH_K2+1, Disabled=FALSE)  // FB1 FB ARITH: Multiplication factor2
        3585 = 3 (Name=ARITH_MODE+1, Disabled=FALSE)  // y = x1 * x2
      ARITH + 2 (Disabled=FALSE)
        3594 = MOTOR_TORQ_RATED (Name=ARITH_IN1_PARID+2, Disabled=FALSE)  // MOTOR_TORQ_RATED -- 53
        3602 = ARITH_VALUE_R4+1 (Name=ARITH_IN2_PARID+2, Disabled=FALSE)  // 3625
        3634 = 0 (Name=ARITH_K1+2, Disabled=FALSE)  // FB2 FB ARITH: Multiplication factor1
        3642 = 0 (Name=ARITH_K2+2, Disabled=FALSE)  // FB2 FB ARITH: Multiplication factor2
        3586 = 1 (Name=ARITH_MODE+2, Disabled=FALSE)  // y = x1 + x2
      ARITH + 3 (Disabled=FALSE)
        3595 = MOTOR_WIND_TEMP_MAX (Name=ARITH_IN1_PARID+3, Disabled=FALSE)  // 74 - MOTOR_WIND_TEMP_MAX
        3603 = TEMP_MOTOR (Name=ARITH_IN2_PARID+3, Disabled=FALSE)  // 381 - TEMP_MOTOR
        3635 = 0 (Name=ARITH_K1+3, Disabled=FALSE)  // FB3 FB ARITH: Multiplication factor1
        3643 = 0 (Name=ARITH_K2+3, Disabled=FALSE)  // FB3 FB ARITH: Multiplication factor2
        3587 = 2 (Name=ARITH_MODE+3, Disabled=FALSE)  // y = x1 - x2
      ARITH + 4 (Disabled=FALSE)
        3596 = ARITH_VALUE_R4+3 (Name=ARITH_IN1_PARID+4, Disabled=FALSE)  // 3627
        3604 = VAR_R4_3+0 (Name=ARITH_IN2_PARID+4, Disabled=FALSE)  // 4152
        3636 = 0 (Name=ARITH_K1+4, Disabled=FALSE)  // FB4 FB ARITH: Multiplication factor1
        3644 = 0 (Name=ARITH_K2+4, Disabled=FALSE)  // FB4 FB ARITH: Multiplication factor2
        3588 = 3 (Name=ARITH_MODE+4, Disabled=FALSE)  // y = x1 * x2
      ARITH + 5 (Disabled=FALSE)
        3597 = MOTOR_TORQ_RATED (Name=ARITH_IN1_PARID+5, Disabled=FALSE)  // MOTOR_TORQ_RATED -- 53
        3605 = ARITH_VALUE_R4+4 (Name=ARITH_IN2_PARID+5, Disabled=FALSE)  // 3628
        3637 = 0 (Name=ARITH_K1+5, Disabled=FALSE)  // FB5 FB ARITH: Multiplication factor1
        3645 = 0 (Name=ARITH_K2+5, Disabled=FALSE)  // FB5 FB ARITH: Multiplication factor2
        3589 = 1 (Name=ARITH_MODE+5, Disabled=FALSE)  // y = x1 + x2
      MINMAX + 0 (Disabled=FALSE)
        12312 = MOTOR_TORQ_MAX (Name=MINMAX_IN1_PARID+0, Disabled=FALSE)  // MOTOR_TORQ_MAX -- 54
        12320 = ARITH_VALUE_R4+2 (Name=MINMAX_IN2_PARID+0, Disabled=FALSE)  // 3626
        12328 = ARITH_VALUE_R4+5 (Name=MINMAX_IN3_PARID+0, Disabled=FALSE)  // 3629
        12288 = 1 (Name=MINMAX_MODE+0, Disabled=FALSE)  // MIN(MOTOR_TORQ_MAX,ARITH_VALUE_R4+1)
      MINMAX + 1 (Disabled=FALSE)
        12313 = VAR_R4_0+0 (Name=MINMAX_IN1_PARID+1, Disabled=FALSE)  // zero
        12321 = MINMAX_VALUE_R4+0 (Name=MINMAX_IN2_PARID+1, Disabled=FALSE)  // FB1 FB MINMAX: Parameter ID of input2
        12289 = 2 (Name=MINMAX_MODE+1, Disabled=FALSE)  // MAX(VAR_R4_0+0,MINMAX_VALUE_R4+0)
      EVWR + 2 (Disabled=FALSE)
        4610 = CONST_I4_ONE (Name=EVWR_EVENT_PARID+2, Disabled=FALSE)  // FB2 FB EVWR: Parameter ID of event input
        4618 = MINMAX_VALUE_R4+1 (Name=EVWR_IN_PARID+2, Disabled=FALSE)  // FB2 FB EVWR: Parameter ID of input
        4626 = 1 (Name=EVWR_EVENT_LEVEL+2, Disabled=FALSE)  // FB2 FB EVWR: Event level
        4634 = LIM_T2_POS (Name=EVWR_WR_PARID+2, Disabled=FALSE)  // 348
        4642 = 2 (Name=EVWR_MODE+2, Disabled=FALSE)  // mode - cyclic write
      EVWR + 3 (Disabled=FALSE)
        4611 = CONST_I4_ONE (Name=EVWR_EVENT_PARID+3, Disabled=FALSE)  // FB3 FB EVWR: Parameter ID of event input
        4619 = MINMAX_VALUE_R4+1 (Name=EVWR_IN_PARID+3, Disabled=FALSE)  // FB3 FB EVWR: Parameter ID of input
        4627 = 1 (Name=EVWR_EVENT_LEVEL+3, Disabled=FALSE)  // FB3 FB EVWR: Event level
        4635 = LIM_T2_NEG (Name=EVWR_WR_PARID+3, Disabled=FALSE)  // 349
        4643 = 2 (Name=EVWR_MODE+3, Disabled=FALSE)  // mode - cyclic write
      EVWR + 4 (Disabled=FALSE)
        4612 = CONST_I4_ONE (Name=EVWR_EVENT_PARID+4, Disabled=FALSE)  // FB4 FB EVWR: Parameter ID of event input
        4620 = MINMAX_VALUE_R4+1 (Name=EVWR_IN_PARID+4, Disabled=FALSE)  // FB4 FB EVWR: Parameter ID of input
        4628 = 1 (Name=EVWR_EVENT_LEVEL+4, Disabled=FALSE)  // FB4 FB EVWR: Event level
        4636 = LIM_T1_POS (Name=EVWR_WR_PARID+4, Disabled=FALSE)  // 248
        4644 = 2 (Name=EVWR_MODE+4, Disabled=FALSE)  // mode - cyclic write
      EVWR + 5 (Disabled=FALSE)
        4613 = CONST_I4_ONE (Name=EVWR_EVENT_PARID+5, Disabled=FALSE)  // FB5 FB EVWR: Parameter ID of event input
        4621 = MINMAX_VALUE_R4+1 (Name=EVWR_IN_PARID+5, Disabled=FALSE)  // FB5 FB EVWR: Parameter ID of input
        4629 = 1 (Name=EVWR_EVENT_LEVEL+5, Disabled=FALSE)  // FB5 FB EVWR: Event level
        4637 = LIM_T1_NEG (Name=EVWR_WR_PARID+5, Disabled=FALSE)  // 249
        4645 = 2 (Name=EVWR_MODE+5, Disabled=FALSE)  // mode - cyclic write
```

### Data object Logical/Motion/para/CarraigeLR (Apt)

#### CarriageLR.apt
```
AcoposParameterTable:
  Root Parameters (Disabled=FALSE)
    Configure Parameter (Disabled=FALSE)
      128 = 1 (Name=SGEN_SW_END_IGNORE, Disabled=FALSE)  // Limit values: Ignore SW end positions
      1196 = 0 (Name=PCTRL_MODE_BITS, Disabled=FALSE)  // CTRL Position controller: Mode bits
      90 = 0 (Name=BRAKE_MODE, Disabled=FALSE)  // Motor holding brake: Mode
      80 = 1 (Name=PHASE_MON_IGNORE, Disabled=FALSE)  // Power mains: Ignore phase failure
      390 = 300 (Name=UDC_NOMINAL, Unit=V, Disabled=FALSE)  // CTRL DC bus: Nominal voltage
    VAR_XX_X+0 (Disabled=FALSE)
      777 = VAR_I4_0+0 (Name=FUNCTION_BLOCK_CREATE, Disabled=FALSE)  // VAR_XX_X+0
      VAR_R4_X_0 (Disabled=FALSE)
        4128 = 0.0 (Name=VAR_R4_0+0, Disabled=FALSE)  // velocity set -- cyclic set
        4136 = 0.0 (Name=VAR_R4_1+0, Disabled=FALSE)  // torque limit -- cyclic set
        4144 = 1.058 (Name=VAR_R4_2+0, Disabled=FALSE)  // temp junction Kp
        4152 = 1.058 (Name=VAR_R4_3+0, Disabled=FALSE)  // temp motor Kp
      VAR_I4_X_0 (Disabled=FALSE)
        4160 = 0.0 (Name=VAR_I2_0+0, Disabled=FALSE)  // FB0 FB VAR: Variable0 I2
        4168 = 0.0 (Name=VAR_I2_1+0, Disabled=FALSE)  // FB0 FB VAR: Variable1 I2
        4176 = 0.0 (Name=VAR_I2_2+0, Disabled=FALSE)  // FB0 FB VAR: Variable2 I2
        4184 = 0.0 (Name=VAR_I2_3+0, Disabled=FALSE)  // FB0 FB VAR: Variable3 I2
    VAR_XX_X+1 (Disabled=FALSE)
      777 = VAR_I4_0+1 (Name=FUNCTION_BLOCK_CREATE, Disabled=FALSE)  // VAR_XX_X+1
      VAR_R4_X_1 (Disabled=FALSE)
        4129 = 0.0 (Name=VAR_R4_0+1, Disabled=FALSE)  // zero
        4137 = 0.0 (Name=VAR_R4_1+1, Disabled=FALSE)  // 288 - SCTRL_ADD_SET_PARID
        4145 = 31 (Name=VAR_R4_2+1, Disabled=FALSE)  // Torque_Max - User Setting
        4153 = 0.0 (Name=VAR_R4_3+1, Disabled=FALSE)  // no use
    VAR_XX_X+2 (Disabled=FALSE)
      777 = VAR_I4_0+2 (Name=FUNCTION_BLOCK_CREATE, Disabled=FALSE)  // VAR_XX_X+2
      VAR_R4_X_2 (Disabled=FALSE)
        4130 = 0.0 (Name=VAR_R4_0+2, Disabled=FALSE)  // Power Consumption Trigger - Left Carriage
        4138 = 0.0 (Name=VAR_R4_1+2, Disabled=FALSE)  // Power Consumption Trigger - Right Carriage
        4146 = 0.0 (Name=VAR_R4_2+2, Disabled=FALSE)  // FB2 FB VAR: Variable2 R4
        4154 = 0.0 (Name=VAR_R4_3+2, Disabled=FALSE)  // FB2 FB VAR: Variable3 R4
    Velocity Control (Disabled=FALSE)
      Function Create (Disabled=FALSE)
        777 = IPL_MODE+0 (Name=FUNCTION_BLOCK_CREATE, Disabled=FALSE)  // IPL_0
        777 = EVWR_MODE+0 (Name=FUNCTION_BLOCK_CREATE, Disabled=FALSE)  // EVWR_0
        777 = CMP_MODE+0 (Name=FUNCTION_BLOCK_CREATE, Disabled=FALSE)  // CMP_0
        777 = EVWR_MODE+1 (Name=FUNCTION_BLOCK_CREATE, Disabled=FALSE)  // EVWR_1
      IPL + 0 (Disabled=FALSE)
        8712 = VAR_R4_0+0 (Name=IPL_IN_PARID+0, Disabled=FALSE)  // velocity set
        8760 = CYCLIC_TODRV_COUNT (Name=IPL_EV_PARID+0, Disabled=FALSE)  // 909 - CYCLIC_TODRV_COUNT
        8720 = 2000 (Name=IPL_CYCLE_TIME+0, Unit=us, Disabled=FALSE)  // FB0 FB IPL: Cycle time
        8728 = 800 (Name=IPL_EXTRAPOLATION_TIME+0, Unit=us, Disabled=FALSE)  // FB0 FB IPL: Extrapolation time
        8704 = 1 (Name=IPL_MODE+0, Disabled=FALSE)  // linear interpolation
      EVWR + 0 (Disabled=FALSE)
        4608 = CMP_VALUE+0 (Name=EVWR_EVENT_PARID+0, Disabled=FALSE)  // v_set == 0
        4616 = IPL_VALUE_R4+0 (Name=EVWR_IN_PARID+0, Disabled=FALSE)  // 8752 -- interpolated v_set
        4624 = 0 (Name=EVWR_EVENT_LEVEL+0, Disabled=FALSE)  // FB0 FB EVWR: Event level
        4632 = VAR_R4_1+1 (Name=EVWR_WR_PARID+0, Disabled=FALSE)  // 288 - SCTRL_ADD_SET_PARID
        4640 = 2 (Name=EVWR_MODE+0, Disabled=FALSE)  // cyclic write
      288 = VAR_R4_1+1 (Name=SCTRL_ADD_SET_PARID, Disabled=FALSE)  // CTRL Speed controller: Parameter ID additive set value
      CMP + 0 (Disabled=FALSE)
        6656 = IPL_VALUE_R4+0 (Name=CMP_IN_PARID+0, Disabled=FALSE)  // 8752 -- interpolated v_set
        6664 = 0 (Name=CMP_THRESHOLD+0, Disabled=FALSE)  // FB0 FB CMP: threshold
        6672 = 0.001 (Name=CMP_WINDOW+0, Disabled=FALSE)  // FB0 FB CMP: window
        6680 = 0 (Name=CMP_HYSTERESIS+0, Disabled=FALSE)  // FB0 FB CMP: hysteresis window
        6688 = 2 (Name=CMP_MODE+0, Disabled=FALSE)  // ==
      231 = CMP_VALUE+0 (Name=PCTRL_ENABLE_PARID, Disabled=FALSE)  // if(interpolated v_set == 0)enable PCTRL
      EVWR + 1 (Disabled=FALSE)
        4609 = CMP_VALUE+0 (Name=EVWR_EVENT_PARID+1, Disabled=FALSE)  // 6696
        4617 = VAR_R4_2+1 (Name=EVWR_IN_PARID+1, Disabled=FALSE)  // FB1 FB EVWR: Parameter ID of input / Torque_Max - User Setting
        4625 = 1 (Name=EVWR_EVENT_LEVEL+1, Disabled=FALSE)  // FB1 FB EVWR: Event level
        4633 = VAR_R4_1+0 (Name=EVWR_WR_PARID+1, Disabled=FALSE)  // FB1 FB EVWR: Parameter ID of output value
        4641 = 2 (Name=EVWR_MODE+1, Disabled=FALSE)  // mode - cyclic write
    Torque Limitation (Disabled=FALSE)
      Function Create (Disabled=FALSE)
        777 = IPL_MODE+1 (Name=FUNCTION_BLOCK_CREATE, Disabled=FALSE)  // IPL_1
        777 = ARITH_MODE+0 (Name=FUNCTION_BLOCK_CREATE, Disabled=FALSE)  // ARITH_0
        777 = ARITH_MODE+1 (Name=FUNCTION_BLOCK_CREATE, Disabled=FALSE)  // ARITH_1
        777 = ARITH_MODE+2 (Name=FUNCTION_BLOCK_CREATE, Disabled=FALSE)  // ARITH_2
        777 = ARITH_MODE+3 (Name=FUNCTION_BLOCK_CREATE, Disabled=FALSE)  // ARITH_3
        777 = ARITH_MODE+4 (Name=FUNCTION_BLOCK_CREATE, Disabled=FALSE)  // ARITH_4
        777 = ARITH_MODE+5 (Name=FUNCTION_BLOCK_CREATE, Disabled=FALSE)  // ARITH_5
        777 = MINMAX_MODE+0 (Name=FUNCTION_BLOCK_CREATE, Disabled=FALSE)  // MINMAX_0
        777 = MINMAX_MODE+1 (Name=FUNCTION_BLOCK_CREATE, Disabled=FALSE)  // MINMAX_1
        777 = EVWR_MODE+2 (Name=FUNCTION_BLOCK_CREATE, Disabled=FALSE)  // EVWR_2
        777 = EVWR_MODE+3 (Name=FUNCTION_BLOCK_CREATE, Disabled=FALSE)  // EVWR_3
        777 = EVWR_MODE+4 (Name=FUNCTION_BLOCK_CREATE, Disabled=FALSE)  // EVWR_4
        777 = EVWR_MODE+5 (Name=FUNCTION_BLOCK_CREATE, Disabled=FALSE)  // EVWR_5
      IPL (Disabled=FALSE)
        8713 = VAR_R4_1+0 (Name=IPL_IN_PARID+1, Disabled=FALSE)  // 4136
        8761 = CYCLIC_TODRV_COUNT (Name=IPL_EV_PARID+1, Disabled=FALSE)  // 909 - CYCLIC_TODRV_COUNT
        8721 = 2000 (Name=IPL_CYCLE_TIME+1, Unit=us, Disabled=FALSE)  // FB1 FB IPL: Cycle time
        8729 = 2000 (Name=IPL_EXTRAPOLATION_TIME+1, Unit=us, Disabled=FALSE)  // FB1 FB IPL: Extrapolation time
        8705 = 1 (Name=IPL_MODE+1, Disabled=FALSE)  // FB1 FB IPL: Mode -- linear interpolation
      ARITH + 0 (Disabled=FALSE)
        3592 = TEMP_JUNCTION_LIM (Name=ARITH_IN1_PARID+0, Disabled=FALSE)  // TEMP_JUNCTION_LIM -- 842
        3600 = TEMP_JUNCTION (Name=ARITH_IN2_PARID+0, Disabled=FALSE)  // TEMP_JUNCTION -- 382
        3632 = 0 (Name=ARITH_K1+0, Disabled=FALSE)  // FB0 FB ARITH: Multiplication factor1
        3640 = 0 (Name=ARITH_K2+0, Disabled=FALSE)  // FB0 FB ARITH: Multiplication factor2
        3584 = 2 (Name=ARITH_MODE+0, Disabled=FALSE)  // y= x1 - x2
      ARITH + 1 (Disabled=FALSE)
        3593 = ARITH_VALUE_R4+0 (Name=ARITH_IN1_PARID+1, Disabled=FALSE)  // 3624
        3601 = VAR_R4_2+0 (Name=ARITH_IN2_PARID+1, Disabled=FALSE)  // 4144
        3633 = 0 (Name=ARITH_K1+1, Disabled=FALSE)  // FB1 FB ARITH: Multiplication factor1
        3641 = 0 (Name=ARITH_K2+1, Disabled=FALSE)  // FB1 FB ARITH: Multiplication factor2
        3585 = 3 (Name=ARITH_MODE+1, Disabled=FALSE)  // y = x1 * x2
      ARITH + 2 (Disabled=FALSE)
        3594 = MOTOR_TORQ_RATED (Name=ARITH_IN1_PARID+2, Disabled=FALSE)  // MOTOR_TORQ_RATED -- 53
        3602 = ARITH_VALUE_R4+1 (Name=ARITH_IN2_PARID+2, Disabled=FALSE)  // 3625
        3634 = 0 (Name=ARITH_K1+2, Disabled=FALSE)  // FB2 FB ARITH: Multiplication factor1
        3642 = 0 (Name=ARITH_K2+2, Disabled=FALSE)  // FB2 FB ARITH: Multiplication factor2
        3586 = 1 (Name=ARITH_MODE+2, Disabled=FALSE)  // y = x1 + x2
      ARITH + 3 (Disabled=FALSE)
        3595 = MOTOR_WIND_TEMP_MAX (Name=ARITH_IN1_PARID+3, Disabled=FALSE)  // 74 - MOTOR_WIND_TEMP_MAX
        3603 = TEMP_MOTOR_MODELL (Name=ARITH_IN2_PARID+3, Disabled=FALSE)  // 393 - TEMP_MOTOR_MODELL
        3635 = 0 (Name=ARITH_K1+3, Disabled=FALSE)  // FB3 FB ARITH: Multiplication factor1
        3643 = 0 (Name=ARITH_K2+3, Disabled=FALSE)  // FB3 FB ARITH: Multiplication factor2
        3587 = 2 (Name=ARITH_MODE+3, Disabled=FALSE)  // y = x1 - x2
      ARITH + 4 (Disabled=FALSE)
        3596 = ARITH_VALUE_R4+3 (Name=ARITH_IN1_PARID+4, Disabled=FALSE)  // 3627
        3604 = VAR_R4_3+0 (Name=ARITH_IN2_PARID+4, Disabled=FALSE)  // 4152
        3636 = 0 (Name=ARITH_K1+4, Disabled=FALSE)  // FB4 FB ARITH: Multiplication factor1
        3644 = 0 (Name=ARITH_K2+4, Disabled=FALSE)  // FB4 FB ARITH: Multiplication factor2
        3588 = 3 (Name=ARITH_MODE+4, Disabled=FALSE)  // y = x1 * x2
      ARITH + 5 (Disabled=FALSE)
        3597 = MOTOR_TORQ_RATED (Name=ARITH_IN1_PARID+5, Disabled=FALSE)  // MOTOR_TORQ_RATED -- 53
        3605 = ARITH_VALUE_R4+4 (Name=ARITH_IN2_PARID+5, Disabled=FALSE)  // 3628
        3637 = 0 (Name=ARITH_K1+5, Disabled=FALSE)  // FB5 FB ARITH: Multiplication factor1
        3645 = 0 (Name=ARITH_K2+5, Disabled=FALSE)  // FB5 FB ARITH: Multiplication factor2
        3589 = 1 (Name=ARITH_MODE+5, Disabled=FALSE)  // y = x1 + x2
      MINMAX + 0 (Disabled=FALSE)
        12312 = VAR_R4_2+1 (Name=MINMAX_IN1_PARID+0, Disabled=FALSE)  // MOTOR_TORQ_MAX -- 54 / Torque_Max - User Setting
        12320 = ARITH_VALUE_R4+2 (Name=MINMAX_IN2_PARID+0, Disabled=FALSE)  // 3626
        12328 = ARITH_VALUE_R4+5 (Name=MINMAX_IN3_PARID+0, Disabled=FALSE)  // 3629
        12336 = IPL_VALUE_R4+1 (Name=MINMAX_IN4_PARID+0, Disabled=FALSE)  // 8753 -- interpolated torque set
        12288 = 1 (Name=MINMAX_MODE+0, Disabled=FALSE)  // MIN(MOTOR_TORQ_MAX,ARITH_VALUE_R4+1)
      MINMAX + 1 (Disabled=FALSE)
        12313 = VAR_R4_0+1 (Name=MINMAX_IN1_PARID+1, Disabled=FALSE)  // zero
        12321 = MINMAX_VALUE_R4+0 (Name=MINMAX_IN2_PARID+1, Disabled=FALSE)  // FB1 FB MINMAX: Parameter ID of input2
        12289 = 2 (Name=MINMAX_MODE+1, Disabled=FALSE)  // MAX(VAR_R4_0+1,MINMAX_VALUE_R4+0)
      EVWR + 2 (Disabled=FALSE)
        4610 = CONST_I4_ONE (Name=EVWR_EVENT_PARID+2, Disabled=FALSE)  // FB2 FB EVWR: Parameter ID of event input
        4618 = MINMAX_VALUE_R4+1 (Name=EVWR_IN_PARID+2, Disabled=FALSE)  // FB2 FB EVWR: Parameter ID of input
        4626 = 1 (Name=EVWR_EVENT_LEVEL+2, Disabled=FALSE)  // FB2 FB EVWR: Event level
        4634 = LIM_T2_POS (Name=EVWR_WR_PARID+2, Disabled=FALSE)  // 348
        4642 = 2 (Name=EVWR_MODE+2, Disabled=FALSE)  // mode - cyclic write
      EVWR + 3 (Disabled=FALSE)
        4611 = CONST_I4_ONE (Name=EVWR_EVENT_PARID+3, Disabled=FALSE)  // FB3 FB EVWR: Parameter ID of event input
        4619 = MINMAX_VALUE_R4+1 (Name=EVWR_IN_PARID+3, Disabled=FALSE)  // FB3 FB EVWR: Parameter ID of input
        4627 = 1 (Name=EVWR_EVENT_LEVEL+3, Disabled=FALSE)  // FB3 FB EVWR: Event level
        4635 = LIM_T2_NEG (Name=EVWR_WR_PARID+3, Disabled=FALSE)  // 349
        4643 = 2 (Name=EVWR_MODE+3, Disabled=FALSE)  // mode - cyclic write
      EVWR + 4 (Disabled=FALSE)
        4612 = CONST_I4_ONE (Name=EVWR_EVENT_PARID+4, Disabled=FALSE)  // FB4 FB EVWR: Parameter ID of event input
        4620 = MINMAX_VALUE_R4+1 (Name=EVWR_IN_PARID+4, Disabled=FALSE)  // FB4 FB EVWR: Parameter ID of input
        4628 = 1 (Name=EVWR_EVENT_LEVEL+4, Disabled=FALSE)  // FB4 FB EVWR: Event level
        4636 = LIM_T1_POS (Name=EVWR_WR_PARID+4, Disabled=FALSE)  // 248
        4644 = 2 (Name=EVWR_MODE+4, Disabled=FALSE)  // mode - cyclic write
      EVWR + 5 (Disabled=FALSE)
        4613 = CONST_I4_ONE (Name=EVWR_EVENT_PARID+5, Disabled=FALSE)  // FB5 FB EVWR: Parameter ID of event input
        4621 = MINMAX_VALUE_R4+1 (Name=EVWR_IN_PARID+5, Disabled=FALSE)  // FB5 FB EVWR: Parameter ID of input
        4629 = 1 (Name=EVWR_EVENT_LEVEL+5, Disabled=FALSE)  // FB5 FB EVWR: Event level
        4637 = LIM_T1_NEG (Name=EVWR_WR_PARID+5, Disabled=FALSE)  // 249
        4645 = 2 (Name=EVWR_MODE+5, Disabled=FALSE)  // mode - cyclic write
    brake resistors (Disabled=TRUE)
      10 = 33 (Name=R_BLEEDER_EXT, Unit=Ohm, Disabled=TRUE)  // Bleeder: External: Resistance
      11 = 637 (Name=TEMP_MAX_BLEEDER_EXT, Unit=°C, Disabled=TRUE)  // Bleeder: External: Limit temperature
      12 = 0.852 (Name=RTH_BLEEDER_AMB_EXT, Unit=K/W, Disabled=TRUE)  // Bleeder: External: Thermal resistance
      13 = 40.68 (Name=CTH_BLEEDER_EXT, Unit=Ws/K, Disabled=TRUE)  // Bleeder: External: Thermal capacity
      398 = 1 (Name=BLEEDER_SELECTOR_EXT, Disabled=TRUE)  // Bleeder: Selector
    8B0W0079H000.000-1 mounting vertical V1 (Disabled=TRUE)
      brake  (Disabled=TRUE)  //  DO NOT USE with ACOPOS Firmware before V2.27.0
      10 = 33 (Name=R_BLEEDER_EXT, Unit=Ohm, Disabled=TRUE)  // Bleeder: External: Resistance
      11 = 673.08 (Name=TEMP_MAX_BLEEDER_EXT, Unit=癈, Disabled=TRUE)  // Bleeder: External: Limit temperature
      12 = 0.852 (Name=RTH_BLEEDER_AMB_EXT, Unit=K/W, Disabled=TRUE)  // Bleeder: External: Thermic resistance
      13 = 40.68 (Name=CTH_BLEEDER_EXT, Unit=Ws/K, Disabled=TRUE)  // Bleeder: External: Thermic capacity
      398 = 1 (Name=BLEEDER_SELECTOR_EXT, Disabled=TRUE)  // Bleeder: Selector
    Power Consumption (Disabled=TRUE)
      1140 = 10000000 (Name=PMET_TIME_IV, Unit=us, Disabled=TRUE)  // PowerMeter: Observation period
      1139 = 1 (Name=PMET_MODE, Disabled=TRUE)  // PowerMeter: Mode
    HardWare Limit  For ACOPOS Multi:
      945 = VAR_I2_0+0 (Name=POS_LIMIT_SWITCH_PARID)  // Digital inputs: Parameter ID for positive end switch
      946 = VAR_I2_1+0 (Name=NEG_LIMIT_SWITCH_PARID)  // Digital inputs: Parameter ID for negative end switch
```

### Data object Logical/Motion/para/BlowPinLR (Apt)

#### BlowPinLR.apt
```
AcoposParameterTable:
  Root Parameters (Disabled=FALSE)
    Configure Parameter (Disabled=FALSE)
      128 = 1 (Name=SGEN_SW_END_IGNORE, Disabled=FALSE)  // Limit values: Ignore SW end positions
      1196 = 0 (Name=PCTRL_MODE_BITS, Disabled=FALSE)  // CTRL Position controller: Mode bits
      80 = 1 (Name=PHASE_MON_IGNORE, Disabled=TRUE)  // Power mains: Ignore phase failure
      300 = 311 (Name=UDC_DETECTION, Unit=V, Disabled=FALSE)  // CTRL DC bus: Voltage detection: Lower limit
      373 = 0 (Name=TEMP_MOTOR_MODEL_MODE)  // Motor: Temperature model: Mode
      1215 = 2 (Name=MOTOR_TEMPSENS_TYPE, Disabled=TRUE)  // Temperature sensor: Type
    VAR_XX_X+0 (Disabled=FALSE)
      777 = VAR_I4_0+0 (Name=FUNCTION_BLOCK_CREATE, Disabled=FALSE)  // VAR_XX_X+0
      VAR_R4_X_0 (Disabled=FALSE)
        4128 = 0.0 (Name=VAR_R4_0+0, Disabled=FALSE)  // velocity set -- cyclic set
        4136 = 0.0 (Name=VAR_R4_1+0, Disabled=FALSE)  // torque limit -- cyclic set
        4144 = 0.666 (Name=VAR_R4_2+0, Disabled=FALSE)  // temp junction Kp
        4152 = 0.666 (Name=VAR_R4_3+0, Disabled=FALSE)  // temp motor Kp
      VAR_R4_X_2 (Disabled=FALSE)
        4160 = 0.0 (Name=VAR_I2_0+0, Disabled=FALSE)  // FB0 FB VAR: Variable0 I2
        4168 = 0.0 (Name=VAR_I2_1+0, Disabled=FALSE)  // FB0 FB VAR: Variable1 I2
        4176 = 0.0 (Name=VAR_I2_2+0, Disabled=FALSE)  // FB0 FB VAR: Variable2 I2
        4184 = 0.0 (Name=VAR_I2_3+0, Disabled=FALSE)  // FB0 FB VAR: Variable3 I2
    VAR_XX_X+1 (Disabled=FALSE)
      777 = VAR_I4_0+1 (Name=FUNCTION_BLOCK_CREATE, Disabled=FALSE)  // VAR_XX_X+1
      VAR_R4_X_1 (Disabled=FALSE)
        4129 = 0.0 (Name=VAR_R4_0+1, Disabled=FALSE)  // zero
        4137 = 0.0 (Name=VAR_R4_1+1, Disabled=FALSE)  // 288 - SCTRL_ADD_SET_PARID
        4145 = 0.0 (Name=VAR_R4_2+1, Disabled=FALSE)  // no use
        4153 = 0.0 (Name=VAR_R4_3+1, Disabled=FALSE)  // no use
    VAR_XX_X+2 (Disabled=FALSE)
      777 = VAR_I4_0+2 (Name=FUNCTION_BLOCK_CREATE, Disabled=FALSE)  // VAR_XX_X+3
      VAR_R4_X_2 (Disabled=FALSE)
        4130 = 0.0 (Name=VAR_R4_0+2, Disabled=FALSE)  // Power Consumption Trigger - Left Carriage
        4138 = 0.0 (Name=VAR_R4_1+2, Disabled=FALSE)  // Power Consumption Trigger - Right Carriage
        4146 = 0.0 (Name=VAR_R4_2+2, Disabled=FALSE)  // FB2 FB VAR: Variable2 R4
        4154 = 0.0 (Name=VAR_R4_3+2, Disabled=FALSE)  // FB2 FB VAR: Variable3 R4
    Velocity Control (Disabled=FALSE)
      Function Create (Disabled=FALSE)
        777 = IPL_MODE+0 (Name=FUNCTION_BLOCK_CREATE, Disabled=FALSE)  // IPL_0
        777 = EVWR_MODE+0 (Name=FUNCTION_BLOCK_CREATE, Disabled=FALSE)  // EVWR_0
        777 = CMP_MODE+0 (Name=FUNCTION_BLOCK_CREATE, Disabled=FALSE)  // CMP_0
        777 = EVWR_MODE+1 (Name=FUNCTION_BLOCK_CREATE, Disabled=FALSE)  // EVWR_1
      IPL + 0 (Disabled=FALSE)
        8712 = VAR_R4_0+0 (Name=IPL_IN_PARID+0, Disabled=FALSE)  // velocity set
        8760 = CYCLIC_TODRV_COUNT (Name=IPL_EV_PARID+0, Disabled=FALSE)  // 909 - CYCLIC_TODRV_COUNT
        8720 = 2000 (Name=IPL_CYCLE_TIME+0, Unit=us, Disabled=FALSE)  // FB0 FB IPL: Cycle time
        8728 = 800 (Name=IPL_EXTRAPOLATION_TIME+0, Unit=us, Disabled=FALSE)  // FB0 FB IPL: Extrapolation time
        8704 = 1 (Name=IPL_MODE+0, Disabled=FALSE)  // linear interpolation
      EVWR + 0 (Disabled=FALSE)
        4608 = CMP_VALUE+0 (Name=EVWR_EVENT_PARID+0, Disabled=FALSE)  // v_set == 0
        4616 = IPL_VALUE_R4+0 (Name=EVWR_IN_PARID+0, Disabled=FALSE)  // 8752 -- interpolated v_set
        4624 = 0 (Name=EVWR_EVENT_LEVEL+0, Disabled=FALSE)  // FB0 FB EVWR: Event level
        4632 = VAR_R4_1+1 (Name=EVWR_WR_PARID+0, Disabled=FALSE)  // 288-SCTRL_ADD_SET_PARID
        4640 = 2 (Name=EVWR_MODE+0, Disabled=FALSE)  // cyclic write
      288 = VAR_R4_1+1 (Name=SCTRL_ADD_SET_PARID, Disabled=FALSE)  // CTRL Speed controller: Parameter ID additive set value
      CMP + 0 (Disabled=FALSE)
        6656 = IPL_VALUE_R4+0 (Name=CMP_IN_PARID+0, Disabled=FALSE)  // 8752 -- interpolated v_set
        6664 = 0 (Name=CMP_THRESHOLD+0, Disabled=FALSE)  // FB0 FB CMP: threshold
        6672 = 0.001 (Name=CMP_WINDOW+0, Disabled=FALSE)  // FB0 FB CMP: window
        6680 = 0 (Name=CMP_HYSTERESIS+0, Disabled=FALSE)  // FB0 FB CMP: hysteresis window
        6688 = 2 (Name=CMP_MODE+0, Disabled=FALSE)  // ==
      231 = CMP_VALUE+0 (Name=PCTRL_ENABLE_PARID, Disabled=FALSE)  // if(interpolated v_set == 0)enable PCTRL
      EVWR + 1 (Disabled=FALSE)
        4609 = CMP_VALUE+0 (Name=EVWR_EVENT_PARID+1, Disabled=FALSE)  // 6696
        4617 = MOTOR_TORQ_MAX (Name=EVWR_IN_PARID+1, Disabled=FALSE)  // FB1 FB EVWR: Parameter ID of input
        4625 = 1 (Name=EVWR_EVENT_LEVEL+1, Disabled=FALSE)  // FB1 FB EVWR: Event level
        4633 = VAR_R4_1+0 (Name=EVWR_WR_PARID+1, Disabled=FALSE)  // FB1 FB EVWR: Parameter ID of output value
        4641 = 2 (Name=EVWR_MODE+1, Disabled=FALSE)  // mode - cyclic write
    Torque Limitation (Disabled=FALSE)
      Function Create (Disabled=FALSE)
        777 = IPL_MODE+1 (Name=FUNCTION_BLOCK_CREATE, Disabled=FALSE)  // IPL_1
        777 = ARITH_MODE+0 (Name=FUNCTION_BLOCK_CREATE, Disabled=FALSE)  // ARITH_0
        777 = ARITH_MODE+1 (Name=FUNCTION_BLOCK_CREATE, Disabled=FALSE)  // ARITH_1
        777 = ARITH_MODE+2 (Name=FUNCTION_BLOCK_CREATE, Disabled=FALSE)  // ARITH_2
        777 = ARITH_MODE+3 (Name=FUNCTION_BLOCK_CREATE, Disabled=FALSE)  // ARITH_3
        777 = ARITH_MODE+4 (Name=FUNCTION_BLOCK_CREATE, Disabled=FALSE)  // ARITH_4
        777 = ARITH_MODE+5 (Name=FUNCTION_BLOCK_CREATE, Disabled=FALSE)  // ARITH_5
        777 = MINMAX_MODE+0 (Name=FUNCTION_BLOCK_CREATE, Disabled=FALSE)  // MINMAX_0
        777 = MINMAX_MODE+1 (Name=FUNCTION_BLOCK_CREATE, Disabled=FALSE)  // MINMAX_1
        777 = EVWR_MODE+2 (Name=FUNCTION_BLOCK_CREATE, Disabled=FALSE)  // EVWR_2
        777 = EVWR_MODE+3 (Name=FUNCTION_BLOCK_CREATE, Disabled=FALSE)  // EVWR_3
        777 = EVWR_MODE+4 (Name=FUNCTION_BLOCK_CREATE, Disabled=FALSE)  // EVWR_4
        777 = EVWR_MODE+5 (Name=FUNCTION_BLOCK_CREATE, Disabled=FALSE)  // EVWR_5
      IPL (Disabled=FALSE)
        8713 = VAR_R4_1+0 (Name=IPL_IN_PARID+1, Disabled=FALSE)  // 4136
        8761 = CYCLIC_TODRV_COUNT (Name=IPL_EV_PARID+1, Disabled=FALSE)  // 909 - CYCLIC_TODRV_COUNT
        8721 = 2000 (Name=IPL_CYCLE_TIME+1, Unit=us, Disabled=FALSE)  // FB1 FB IPL: Cycle time
        8729 = 2000 (Name=IPL_EXTRAPOLATION_TIME+1, Unit=us, Disabled=FALSE)  // FB1 FB IPL: Extrapolation time
        8705 = 1 (Name=IPL_MODE+1, Disabled=FALSE)  // FB1 FB IPL: Mode -- linear interpolation
      ARITH + 0 (Disabled=FALSE)
        3592 = TEMP_JUNCTION_LIM (Name=ARITH_IN1_PARID+0, Disabled=FALSE)  // TEMP_JUNCTION_LIM -- 842
        3600 = TEMP_JUNCTION (Name=ARITH_IN2_PARID+0, Disabled=FALSE)  // TEMP_JUNCTION -- 382
        3632 = 0 (Name=ARITH_K1+0, Disabled=FALSE)  // FB0 FB ARITH: Multiplication factor1
        3640 = 0 (Name=ARITH_K2+0, Disabled=FALSE)  // FB0 FB ARITH: Multiplication factor2
        3584 = 2 (Name=ARITH_MODE+0, Disabled=FALSE)  // y= x1 - x2
      ARITH + 1 (Disabled=FALSE)
        3593 = ARITH_VALUE_R4+0 (Name=ARITH_IN1_PARID+1, Disabled=FALSE)  // 3624
        3601 = VAR_R4_2+0 (Name=ARITH_IN2_PARID+1, Disabled=FALSE)  // 4144
        3633 = 0 (Name=ARITH_K1+1, Disabled=FALSE)  // FB1 FB ARITH: Multiplication factor1
        3641 = 0 (Name=ARITH_K2+1, Disabled=FALSE)  // FB1 FB ARITH: Multiplication factor2
        3585 = 3 (Name=ARITH_MODE+1, Disabled=FALSE)  // y = x1 * x2
      ARITH + 2 (Disabled=FALSE)
        3594 = MOTOR_TORQ_RATED (Name=ARITH_IN1_PARID+2, Disabled=FALSE)  // MOTOR_TORQ_RATED -- 53
        3602 = ARITH_VALUE_R4+1 (Name=ARITH_IN2_PARID+2, Disabled=FALSE)  // 3625
        3634 = 0 (Name=ARITH_K1+2, Disabled=FALSE)  // FB2 FB ARITH: Multiplication factor1
        3642 = 0 (Name=ARITH_K2+2, Disabled=FALSE)  // FB2 FB ARITH: Multiplication factor2
        3586 = 1 (Name=ARITH_MODE+2, Disabled=FALSE)  // y = x1 + x2
      ARITH + 3 (Disabled=FALSE)
        3595 = MOTOR_WIND_TEMP_MAX (Name=ARITH_IN1_PARID+3, Disabled=FALSE)  // 74 - MOTOR_WIND_TEMP_MAX
        3603 = TEMP_MOTOR_MODELL (Name=ARITH_IN2_PARID+3, Disabled=FALSE)  // 393 - TEMP_MOTOR_MODELL
        3635 = 0 (Name=ARITH_K1+3, Disabled=FALSE)  // FB3 FB ARITH: Multiplication factor1
        3643 = 0 (Name=ARITH_K2+3, Disabled=FALSE)  // FB3 FB ARITH: Multiplication factor2
        3587 = 2 (Name=ARITH_MODE+3, Disabled=FALSE)  // y = x1 - x2
      ARITH + 4 (Disabled=FALSE)
        3596 = ARITH_VALUE_R4+3 (Name=ARITH_IN1_PARID+4, Disabled=FALSE)  // 3627
        3604 = VAR_R4_3+0 (Name=ARITH_IN2_PARID+4, Disabled=FALSE)  // 4152
        3636 = 0 (Name=ARITH_K1+4, Disabled=FALSE)  // FB4 FB ARITH: Multiplication factor1
        3644 = 0 (Name=ARITH_K2+4, Disabled=FALSE)  // FB4 FB ARITH: Multiplication factor2
        3588 = 3 (Name=ARITH_MODE+4, Disabled=FALSE)  // y = x1 * x2
      ARITH + 5 (Disabled=FALSE)
        3597 = MOTOR_TORQ_RATED (Name=ARITH_IN1_PARID+5, Disabled=FALSE)  // MOTOR_TORQ_RATED -- 53
        3605 = ARITH_VALUE_R4+4 (Name=ARITH_IN2_PARID+5, Disabled=FALSE)  // 3628
        3637 = 0 (Name=ARITH_K1+5, Disabled=FALSE)  // FB5 FB ARITH: Multiplication factor1
        3645 = 0 (Name=ARITH_K2+5, Disabled=FALSE)  // FB5 FB ARITH: Multiplication factor2
        3589 = 1 (Name=ARITH_MODE+5, Disabled=FALSE)  // y = x1 + x2
      MINMAX + 0 (Disabled=FALSE)
        12312 = MOTOR_TORQ_MAX (Name=MINMAX_IN1_PARID+0, Disabled=FALSE)  // MOTOR_TORQ_MAX -- 54
        12320 = ARITH_VALUE_R4+2 (Name=MINMAX_IN2_PARID+0, Disabled=FALSE)  // 3626
        12328 = ARITH_VALUE_R4+5 (Name=MINMAX_IN3_PARID+0, Disabled=FALSE)  // 3629
        12336 = IPL_VALUE_R4+1 (Name=MINMAX_IN4_PARID+0, Disabled=FALSE)  // 8753 -- interpolated torque set
        12288 = 1 (Name=MINMAX_MODE+0, Disabled=FALSE)  // MIN(MOTOR_TORQ_MAX,ARITH_VALUE_R4+1)
      MINMAX + 1 (Disabled=FALSE)
        12313 = VAR_R4_0+1 (Name=MINMAX_IN1_PARID+1, Disabled=FALSE)  // zero
        12321 = MINMAX_VALUE_R4+0 (Name=MINMAX_IN2_PARID+1, Disabled=FALSE)  // FB1 FB MINMAX: Parameter ID of input2
        12289 = 2 (Name=MINMAX_MODE+1, Disabled=FALSE)  // MAX(VAR_R4_0+1,MINMAX_VALUE_R4+0)
      EVWR + 2 (Disabled=FALSE)
        4610 = CONST_I4_ONE (Name=EVWR_EVENT_PARID+2, Disabled=FALSE)  // FB2 FB EVWR: Parameter ID of event input
        4618 = MINMAX_VALUE_R4+1 (Name=EVWR_IN_PARID+2, Disabled=FALSE)  // FB2 FB EVWR: Parameter ID of input
        4626 = 1 (Name=EVWR_EVENT_LEVEL+2, Disabled=FALSE)  // FB2 FB EVWR: Event level
        4634 = LIM_T2_POS (Name=EVWR_WR_PARID+2, Disabled=FALSE)  // 348
        4642 = 2 (Name=EVWR_MODE+2, Disabled=FALSE)  // mode - cyclic write
      EVWR + 3 (Disabled=FALSE)
        4611 = CONST_I4_ONE (Name=EVWR_EVENT_PARID+3, Disabled=FALSE)  // FB3 FB EVWR: Parameter ID of event input
        4619 = MINMAX_VALUE_R4+1 (Name=EVWR_IN_PARID+3, Disabled=FALSE)  // FB3 FB EVWR: Parameter ID of input
        4627 = 1 (Name=EVWR_EVENT_LEVEL+3, Disabled=FALSE)  // FB3 FB EVWR: Event level
        4635 = LIM_T2_NEG (Name=EVWR_WR_PARID+3, Disabled=FALSE)  // 349
        4643 = 2 (Name=EVWR_MODE+3, Disabled=FALSE)  // mode - cyclic write
      EVWR + 4 (Disabled=FALSE)
        4612 = CONST_I4_ONE (Name=EVWR_EVENT_PARID+4, Disabled=FALSE)  // FB4 FB EVWR: Parameter ID of event input
        4620 = MINMAX_VALUE_R4+1 (Name=EVWR_IN_PARID+4, Disabled=FALSE)  // FB4 FB EVWR: Parameter ID of input
        4628 = 1 (Name=EVWR_EVENT_LEVEL+4, Disabled=FALSE)  // FB4 FB EVWR: Event level
        4636 = LIM_T1_POS (Name=EVWR_WR_PARID+4, Disabled=FALSE)  // 248
        4644 = 2 (Name=EVWR_MODE+4, Disabled=FALSE)  // mode - cyclic write
      EVWR + 5 (Disabled=FALSE)
        4613 = CONST_I4_ONE (Name=EVWR_EVENT_PARID+5, Disabled=FALSE)  // FB5 FB EVWR: Parameter ID of event input
        4621 = MINMAX_VALUE_R4+1 (Name=EVWR_IN_PARID+5, Disabled=FALSE)  // FB5 FB EVWR: Parameter ID of input
        4629 = 1 (Name=EVWR_EVENT_LEVEL+5, Disabled=FALSE)  // FB5 FB EVWR: Event level
        4637 = LIM_T1_NEG (Name=EVWR_WR_PARID+5, Disabled=FALSE)  // 249
        4645 = 2 (Name=EVWR_MODE+5, Disabled=FALSE)  // mode - cyclic write
    HardWare Limit  For ACOPOS Multi:
      945 = VAR_I2_0+0 (Name=POS_LIMIT_SWITCH_PARID)  // Digital inputs: Parameter ID for positive end switch
      946 = VAR_I2_1+0 (Name=NEG_LIMIT_SWITCH_PARID)  // Digital inputs: Parameter ID for negative end switch
```

### Data object Logical/Motion/para/Power (Apt)

#### Power.apt
```
AcoposParameterTable:
  Root Parameters:
    8B0W0079H000.000-1 mounting vertical V1 (Disabled=FALSE)  // Reference: Series and parallel connection of braking resistors 
      brake  (Disabled=FALSE)  //  DO NOT USE with ACOPOS Firmware before V2.27.0
      10 = 11 (Name=R_BLEEDER_EXT, Unit=Ohm, Disabled=FALSE)  // Bleeder: External: Resistance
      12 = 0.284 (Name=RTH_BLEEDER_AMB_EXT, Unit=K/W, Disabled=FALSE)  // Bleeder: External: Thermic resistance
      11 = 670 (Name=TEMP_MAX_BLEEDER_EXT, Unit=H, Disabled=FALSE)  // Bleeder: External: Limit temperature
      13 = 122.04 (Name=CTH_BLEEDER_EXT, Unit=Ws/K, Disabled=FALSE)  // Bleeder: External: Thermic capacity
      398 = 1 (Name=BLEEDER_SELECTOR_EXT, Disabled=FALSE)  // Bleeder: Selector
```

### Data object Logical/Motion/para/nBlowPinLR (Apt)

#### nBlowPinLR.apt
```
AcoposParameterTable:
  Root Parameters (Disabled=FALSE)
    Configure Parameter (Disabled=FALSE)
      128 = 1 (Name=SGEN_SW_END_IGNORE, Disabled=FALSE)  // Limit values: Ignore SW end positions
      1196 = 0 (Name=PCTRL_MODE_BITS, Disabled=FALSE)  // CTRL Position controller: Mode bits
      80 = 1 (Name=PHASE_MON_IGNORE, Disabled=FALSE)  // Power mains: Ignore phase failure
      300 = 311 (Name=UDC_DETECTION, Unit=V, Disabled=FALSE)  // CTRL DC bus: Voltage detection: Lower limit
    VAR_XX_X+0 (Disabled=FALSE)
      777 = VAR_I4_0+0 (Name=FUNCTION_BLOCK_CREATE, Disabled=FALSE)  // VAR_XX_X+0
      VAR_R4_X_0 (Disabled=FALSE)
        4128 = 0.0 (Name=VAR_R4_0+0, Disabled=FALSE)  // velocity set -- cyclic set
        4136 = 0.0 (Name=VAR_R4_1+0, Disabled=FALSE)  // torque limit -- cyclic set
        4144 = 0.666 (Name=VAR_R4_2+0, Disabled=FALSE)  // temp junction Kp
        4152 = 0.666 (Name=VAR_R4_3+0, Disabled=FALSE)  // temp motor Kp
    VAR_XX_X+1 (Disabled=FALSE)
      777 = VAR_I4_0+1 (Name=FUNCTION_BLOCK_CREATE, Disabled=FALSE)  // VAR_XX_X+1
      VAR_R4_X_1 (Disabled=FALSE)
        4129 = 0.0 (Name=VAR_R4_0+1, Disabled=FALSE)  // zero
        4137 = 0.0 (Name=VAR_R4_1+1, Disabled=FALSE)  // 288 - SCTRL_ADD_SET_PARID
        4145 = 0.0 (Name=VAR_R4_2+1, Disabled=FALSE)  // no use
        4153 = 0.0 (Name=VAR_R4_3+1, Disabled=FALSE)  // no use
    VAR_XX_X+3 (Disabled=FALSE)
      777 = VAR_I4_0+3 (Name=FUNCTION_BLOCK_CREATE, Disabled=FALSE)  // VAR_XX_X+3
      VAR_R4_X_2 (Disabled=FALSE)
        4160 = 0.0 (Name=VAR_I2_0+0, Disabled=FALSE)  // FB0 FB VAR: Variable0 I2
        4168 = 0.0 (Name=VAR_I2_1+0, Disabled=FALSE)  // FB0 FB VAR: Variable1 I2
        4176 = 0.0 (Name=VAR_I2_2+0, Disabled=FALSE)  // FB0 FB VAR: Variable2 I2
        4184 = 0.0 (Name=VAR_I2_3+0, Disabled=FALSE)  // FB0 FB VAR: Variable3 I2
    Velocity Control (Disabled=FALSE)
      Function Create (Disabled=FALSE)
        777 = IPL_MODE+0 (Name=FUNCTION_BLOCK_CREATE, Disabled=FALSE)  // IPL_0
        777 = EVWR_MODE+0 (Name=FUNCTION_BLOCK_CREATE, Disabled=FALSE)  // EVWR_0
        777 = CMP_MODE+0 (Name=FUNCTION_BLOCK_CREATE, Disabled=FALSE)  // CMP_0
        777 = EVWR_MODE+1 (Name=FUNCTION_BLOCK_CREATE, Disabled=FALSE)  // EVWR_1
        777 = ARITH_MODE+6 (Name=FUNCTION_BLOCK_CREATE, Disabled=FALSE)  // EVWR_6
        777 = ARITH_MODE+7 (Name=FUNCTION_BLOCK_CREATE, Disabled=FALSE)  // EVWR_7
      IPL + 0 (Disabled=FALSE)
        8712 = VAR_R4_0+0 (Name=IPL_IN_PARID+0, Disabled=FALSE)  // velocity set
        8760 = CYCLIC_TODRV_COUNT (Name=IPL_EV_PARID+0, Disabled=FALSE)  // 909 - CYCLIC_TODRV_COUNT
        8720 = 2000 (Name=IPL_CYCLE_TIME+0, Unit=us, Disabled=FALSE)  // FB0 FB IPL: Cycle time
        8728 = 800 (Name=IPL_EXTRAPOLATION_TIME+0, Unit=us, Disabled=FALSE)  // FB0 FB IPL: Extrapolation time
        8704 = 1 (Name=IPL_MODE+0, Disabled=FALSE)  // linear interpolation
      EVWR + 0 (Disabled=FALSE)
        4608 = CMP_VALUE+0 (Name=EVWR_EVENT_PARID+0, Disabled=FALSE)  // v_set == 0
        4616 = IPL_VALUE_R4+0 (Name=EVWR_IN_PARID+0, Disabled=FALSE)  // 8752 -- interpolated v_set
        4624 = 0 (Name=EVWR_EVENT_LEVEL+0, Disabled=FALSE)  // FB0 FB EVWR: Event level
        4632 = VAR_R4_1+1 (Name=EVWR_WR_PARID+0, Disabled=FALSE)  // 288-SCTRL_ADD_SET_PARID
        4640 = 2 (Name=EVWR_MODE+0, Disabled=FALSE)  // cyclic write
      ARITH + 6 (Disabled=FALSE)
        3598 = VCTRL_SCALE_LOAD_UNITS (Name=ARITH_IN1_PARID+6, Disabled=FALSE)  // FB6 FB ARITH: Parameter ID of input1
        3606 = VCTRL_SCALE_LOAD_MOTREV (Name=ARITH_IN2_PARID+6, Disabled=FALSE)  // FB6 FB ARITH: Parameter ID of input2
        3638 = 0 (Name=ARITH_K1+6, Disabled=FALSE)  // FB6 FB ARITH: Multiplication factor1
        3646 = 0 (Name=ARITH_K2+6, Disabled=FALSE)  // FB6 FB ARITH: Multiplication factor2
        3590 = 5 (Name=ARITH_MODE+6, Disabled=FALSE)  // FB6 FB ARITH: Mode
      ARITH + 7 (Disabled=FALSE)
        3599 = VAR_R4_1+1 (Name=ARITH_IN1_PARID+7, Disabled=FALSE)  // FB7 FB ARITH: Parameter ID of input1
        3607 = ARITH_VALUE_R4+6 (Name=ARITH_IN2_PARID+7, Disabled=FALSE)  // FB7 FB ARITH: Parameter ID of input2
        3639 = 0 (Name=ARITH_K1+7, Disabled=FALSE)  // FB7 FB ARITH: Multiplication factor1
        3647 = 0 (Name=ARITH_K2+7, Disabled=FALSE)  // FB7 FB ARITH: Multiplication factor2
        3591 = 5 (Name=ARITH_MODE+7, Disabled=FALSE)  // FB7 FB ARITH: Mode
      288 = ARITH_VALUE_R4+7 (Name=SCTRL_ADD_SET_PARID, Disabled=FALSE)  // CTRL Speed controller: Parameter ID additive set value
      CMP + 0 (Disabled=FALSE)
        6656 = IPL_VALUE_R4+0 (Name=CMP_IN_PARID+0, Disabled=FALSE)  // 8752 -- interpolated v_set
        6664 = 0 (Name=CMP_THRESHOLD+0, Disabled=FALSE)  // FB0 FB CMP: threshold
        6672 = 0.001 (Name=CMP_WINDOW+0, Disabled=FALSE)  // FB0 FB CMP: window
        6680 = 0 (Name=CMP_HYSTERESIS+0, Disabled=FALSE)  // FB0 FB CMP: hysteresis window
        6688 = 2 (Name=CMP_MODE+0, Disabled=FALSE)  // ==
      231 = CMP_VALUE+0 (Name=PCTRL_ENABLE_PARID, Disabled=FALSE)  // if(interpolated v_set == 0)enable PCTRL
      EVWR + 1 (Disabled=FALSE)
        4609 = CMP_VALUE+0 (Name=EVWR_EVENT_PARID+1, Disabled=FALSE)  // 6696
        4617 = MOTOR_TORQ_MAX (Name=EVWR_IN_PARID+1, Disabled=FALSE)  // FB1 FB EVWR: Parameter ID of input
        4625 = 1 (Name=EVWR_EVENT_LEVEL+1, Disabled=FALSE)  // FB1 FB EVWR: Event level
        4633 = VAR_R4_1+0 (Name=EVWR_WR_PARID+1, Disabled=FALSE)  // FB1 FB EVWR: Parameter ID of output value
        4641 = 2 (Name=EVWR_MODE+1, Disabled=FALSE)  // mode - cyclic write
    Torque Limitation (Disabled=FALSE)
      Function Create (Disabled=FALSE)
        777 = IPL_MODE+1 (Name=FUNCTION_BLOCK_CREATE, Disabled=FALSE)  // IPL_1
        777 = ARITH_MODE+0 (Name=FUNCTION_BLOCK_CREATE, Disabled=FALSE)  // ARITH_0
        777 = ARITH_MODE+1 (Name=FUNCTION_BLOCK_CREATE, Disabled=FALSE)  // ARITH_1
        777 = ARITH_MODE+2 (Name=FUNCTION_BLOCK_CREATE, Disabled=FALSE)  // ARITH_2
        777 = ARITH_MODE+3 (Name=FUNCTION_BLOCK_CREATE, Disabled=FALSE)  // ARITH_3
        777 = ARITH_MODE+4 (Name=FUNCTION_BLOCK_CREATE, Disabled=FALSE)  // ARITH_4
        777 = ARITH_MODE+5 (Name=FUNCTION_BLOCK_CREATE, Disabled=FALSE)  // ARITH_5
        777 = MINMAX_MODE+0 (Name=FUNCTION_BLOCK_CREATE, Disabled=FALSE)  // MINMAX_0
        777 = MINMAX_MODE+1 (Name=FUNCTION_BLOCK_CREATE, Disabled=FALSE)  // MINMAX_1
        777 = EVWR_MODE+2 (Name=FUNCTION_BLOCK_CREATE, Disabled=FALSE)  // EVWR_2
        777 = EVWR_MODE+3 (Name=FUNCTION_BLOCK_CREATE, Disabled=FALSE)  // EVWR_3
        777 = EVWR_MODE+4 (Name=FUNCTION_BLOCK_CREATE, Disabled=FALSE)  // EVWR_4
        777 = EVWR_MODE+5 (Name=FUNCTION_BLOCK_CREATE, Disabled=FALSE)  // EVWR_5
      IPL (Disabled=FALSE)
        8713 = VAR_R4_1+0 (Name=IPL_IN_PARID+1, Disabled=FALSE)  // 4136
        8761 = CYCLIC_TODRV_COUNT (Name=IPL_EV_PARID+1, Disabled=FALSE)  // 909 - CYCLIC_TODRV_COUNT
        8721 = 2000 (Name=IPL_CYCLE_TIME+1, Unit=us, Disabled=FALSE)  // FB1 FB IPL: Cycle time
        8729 = 2000 (Name=IPL_EXTRAPOLATION_TIME+1, Unit=us, Disabled=FALSE)  // FB1 FB IPL: Extrapolation time
        8705 = 1 (Name=IPL_MODE+1, Disabled=FALSE)  // FB1 FB IPL: Mode -- linear interpolation
      ARITH + 0 (Disabled=FALSE)
        3592 = TEMP_JUNCTION_LIM (Name=ARITH_IN1_PARID+0, Disabled=FALSE)  // TEMP_JUNCTION_LIM -- 842
        3600 = TEMP_JUNCTION (Name=ARITH_IN2_PARID+0, Disabled=FALSE)  // TEMP_JUNCTION -- 382
        3632 = 0 (Name=ARITH_K1+0, Disabled=FALSE)  // FB0 FB ARITH: Multiplication factor1
        3640 = 0 (Name=ARITH_K2+0, Disabled=FALSE)  // FB0 FB ARITH: Multiplication factor2
        3584 = 2 (Name=ARITH_MODE+0, Disabled=FALSE)  // y= x1 - x2
      ARITH + 1 (Disabled=FALSE)
        3593 = ARITH_VALUE_R4+0 (Name=ARITH_IN1_PARID+1, Disabled=FALSE)  // 3624
        3601 = VAR_R4_2+0 (Name=ARITH_IN2_PARID+1, Disabled=FALSE)  // 4144
        3633 = 0 (Name=ARITH_K1+1, Disabled=FALSE)  // FB1 FB ARITH: Multiplication factor1
        3641 = 0 (Name=ARITH_K2+1, Disabled=FALSE)  // FB1 FB ARITH: Multiplication factor2
        3585 = 3 (Name=ARITH_MODE+1, Disabled=FALSE)  // y = x1 * x2
      ARITH + 2 (Disabled=FALSE)
        3594 = MOTOR_TORQ_RATED (Name=ARITH_IN1_PARID+2, Disabled=FALSE)  // MOTOR_TORQ_RATED -- 53
        3602 = ARITH_VALUE_R4+1 (Name=ARITH_IN2_PARID+2, Disabled=FALSE)  // 3625
        3634 = 0 (Name=ARITH_K1+2, Disabled=FALSE)  // FB2 FB ARITH: Multiplication factor1
        3642 = 0 (Name=ARITH_K2+2, Disabled=FALSE)  // FB2 FB ARITH: Multiplication factor2
        3586 = 1 (Name=ARITH_MODE+2, Disabled=FALSE)  // y = x1 + x2
      ARITH + 3 (Disabled=FALSE)
        3595 = MOTOR_WIND_TEMP_MAX (Name=ARITH_IN1_PARID+3, Disabled=FALSE)  // 74 - MOTOR_WIND_TEMP_MAX
        3603 = TEMP_MOTOR_MODELL (Name=ARITH_IN2_PARID+3, Disabled=FALSE)  // 393 - TEMP_MOTOR_MODELL
        3635 = 0 (Name=ARITH_K1+3, Disabled=FALSE)  // FB3 FB ARITH: Multiplication factor1
        3643 = 0 (Name=ARITH_K2+3, Disabled=FALSE)  // FB3 FB ARITH: Multiplication factor2
        3587 = 2 (Name=ARITH_MODE+3, Disabled=FALSE)  // y = x1 - x2
      ARITH + 4 (Disabled=FALSE)
        3596 = ARITH_VALUE_R4+3 (Name=ARITH_IN1_PARID+4, Disabled=FALSE)  // 3627
        3604 = VAR_R4_3+0 (Name=ARITH_IN2_PARID+4, Disabled=FALSE)  // 4152
        3636 = 0 (Name=ARITH_K1+4, Disabled=FALSE)  // FB4 FB ARITH: Multiplication factor1
        3644 = 0 (Name=ARITH_K2+4, Disabled=FALSE)  // FB4 FB ARITH: Multiplication factor2
        3588 = 3 (Name=ARITH_MODE+4, Disabled=FALSE)  // y = x1 * x2
      ARITH + 5 (Disabled=FALSE)
        3597 = MOTOR_TORQ_RATED (Name=ARITH_IN1_PARID+5, Disabled=FALSE)  // MOTOR_TORQ_RATED -- 53
        3605 = ARITH_VALUE_R4+4 (Name=ARITH_IN2_PARID+5, Disabled=FALSE)  // 3628
        3637 = 0 (Name=ARITH_K1+5, Disabled=FALSE)  // FB5 FB ARITH: Multiplication factor1
        3645 = 0 (Name=ARITH_K2+5, Disabled=FALSE)  // FB5 FB ARITH: Multiplication factor2
        3589 = 1 (Name=ARITH_MODE+5, Disabled=FALSE)  // y = x1 + x2
      MINMAX + 0 (Disabled=FALSE)
        12312 = MOTOR_TORQ_MAX (Name=MINMAX_IN1_PARID+0, Disabled=FALSE)  // MOTOR_TORQ_MAX -- 54
        12320 = ARITH_VALUE_R4+2 (Name=MINMAX_IN2_PARID+0, Disabled=FALSE)  // 3626
        12328 = ARITH_VALUE_R4+5 (Name=MINMAX_IN3_PARID+0, Disabled=FALSE)  // 3629
        12336 = IPL_VALUE_R4+1 (Name=MINMAX_IN4_PARID+0, Disabled=FALSE)  // 8753 -- interpolated torque set
        12288 = 1 (Name=MINMAX_MODE+0, Disabled=FALSE)  // MIN(MOTOR_TORQ_MAX,ARITH_VALUE_R4+1)
      MINMAX + 1 (Disabled=FALSE)
        12313 = VAR_R4_0+1 (Name=MINMAX_IN1_PARID+1, Disabled=FALSE)  // zero
        12321 = MINMAX_VALUE_R4+0 (Name=MINMAX_IN2_PARID+1, Disabled=FALSE)  // FB1 FB MINMAX: Parameter ID of input2
        12289 = 2 (Name=MINMAX_MODE+1, Disabled=FALSE)  // MAX(VAR_R4_0+1,MINMAX_VALUE_R4+0)
      EVWR + 2 (Disabled=FALSE)
        4610 = CONST_I4_ONE (Name=EVWR_EVENT_PARID+2, Disabled=FALSE)  // FB2 FB EVWR: Parameter ID of event input
        4618 = MINMAX_VALUE_R4+1 (Name=EVWR_IN_PARID+2, Disabled=FALSE)  // FB2 FB EVWR: Parameter ID of input
        4626 = 1 (Name=EVWR_EVENT_LEVEL+2, Disabled=FALSE)  // FB2 FB EVWR: Event level
        4634 = LIM_T2_POS (Name=EVWR_WR_PARID+2, Disabled=FALSE)  // 348
        4642 = 2 (Name=EVWR_MODE+2, Disabled=FALSE)  // mode - cyclic write
      EVWR + 3 (Disabled=FALSE)
        4611 = CONST_I4_ONE (Name=EVWR_EVENT_PARID+3, Disabled=FALSE)  // FB3 FB EVWR: Parameter ID of event input
        4619 = MINMAX_VALUE_R4+1 (Name=EVWR_IN_PARID+3, Disabled=FALSE)  // FB3 FB EVWR: Parameter ID of input
        4627 = 1 (Name=EVWR_EVENT_LEVEL+3, Disabled=FALSE)  // FB3 FB EVWR: Event level
        4635 = LIM_T2_NEG (Name=EVWR_WR_PARID+3, Disabled=FALSE)  // 349
        4643 = 2 (Name=EVWR_MODE+3, Disabled=FALSE)  // mode - cyclic write
      EVWR + 4 (Disabled=FALSE)
        4612 = CONST_I4_ONE (Name=EVWR_EVENT_PARID+4, Disabled=FALSE)  // FB4 FB EVWR: Parameter ID of event input
        4620 = MINMAX_VALUE_R4+1 (Name=EVWR_IN_PARID+4, Disabled=FALSE)  // FB4 FB EVWR: Parameter ID of input
        4628 = 1 (Name=EVWR_EVENT_LEVEL+4, Disabled=FALSE)  // FB4 FB EVWR: Event level
        4636 = LIM_T1_POS (Name=EVWR_WR_PARID+4, Disabled=FALSE)  // 248
        4644 = 2 (Name=EVWR_MODE+4, Disabled=FALSE)  // mode - cyclic write
      EVWR + 5 (Disabled=FALSE)
        4613 = CONST_I4_ONE (Name=EVWR_EVENT_PARID+5, Disabled=FALSE)  // FB5 FB EVWR: Parameter ID of event input
        4621 = MINMAX_VALUE_R4+1 (Name=EVWR_IN_PARID+5, Disabled=FALSE)  // FB5 FB EVWR: Parameter ID of input
        4629 = 1 (Name=EVWR_EVENT_LEVEL+5, Disabled=FALSE)  // FB5 FB EVWR: Event level
        4637 = LIM_T1_NEG (Name=EVWR_WR_PARID+5, Disabled=FALSE)  // 249
        4645 = 2 (Name=EVWR_MODE+5, Disabled=FALSE)  // mode - cyclic write
    HardWare Limit  For ACOPOS Multi:
      945 = VAR_I2_0+0 (Name=POS_LIMIT_SWITCH_PARID)  // Digital inputs: Parameter ID for positive end switch
      946 = VAR_I2_1+0 (Name=NEG_LIMIT_SWITCH_PARID)  // Digital inputs: Parameter ID for negative end switch
```

### Data object Logical/Motion/para/nCarraigeLR (Apt)
